
// ===== library: MasterCopy "DCS3" =====

VAR_GLOBAL   // PLC tag table "Default tag table"
   "Tag_1" AT %IW64 : Word;
   "Tag_2" AT %IW0 : Word;
   "Tag_3" AT %QW0 : Word;
   "TP_start" AT %I7.3 : Bool;
   "TP_stop" AT %I7.4 : Bool;
   "Fire" AT %I7.5 : Bool;
   "To_open_valve" AT %I7.6 : Bool;
   "Spark_on" AT %I7.7 : Bool;
   "Spark_on_1" AT %I8.0 : Bool;
   "Spark_on_2" AT %I8.1 : Bool;
   "Spark_on_3" AT %I8.2 : Bool;
   "Fire_1" AT %I8.3 : Bool;
   "Fire_2" AT %I8.4 : Bool;
   "Fire_3" AT %I8.5 : Bool;
   "Reserv_word" AT %IW68 : Word;
   "MB_Start" AT %I8.6 : Bool;   // false
   "MB_Stop" AT %I9.1 : Bool;
   "Sim_man" AT %I9.2 : Bool;
   "Sim_P_gaz_low" AT %I9.3 : Bool;
   "Sim_ACP_in" AT %IW70 : Word;
   "test" AT %I9.4 : Bool;
   "P_gaz_low" AT %I9.5 : Bool;
   "test_p_low" AT %I9.6 : Bool;
   "Tag_4" AT %IW96 : Word;
   "Tag_5" AT %IW98 : Word;
   "Clock_Byte" AT %MB0 : Byte;
   "Clock_10Hz" AT %M0.0 : Bool;
   "Clock_5Hz" AT %M0.1 : Bool;
   "Clock_2.5Hz" AT %M0.2 : Bool;
   "Clock_2Hz" AT %M0.3 : Bool;
   "Clock_1.25Hz" AT %M0.4 : Bool;
   "Clock_1Hz" AT %M0.5 : Bool;
   "Clock_0.625Hz" AT %M0.6 : Bool;
   "Clock_0.5Hz" AT %M0.7 : Bool;
   "System_Byte" AT %MB1 : Byte;
   "FirstScan" AT %M1.0 : Bool;
   "DiagStatusUpdate" AT %M1.1 : Bool;
   "AlwaysTRUE" AT %M1.2 : Bool;
   "AlwaysFALSE" AT %M1.3 : Bool;
END_VAR

TYPE "dt_AI"
   STRUCT
      Acp : DInt;   // Actual ADC code
      State : Word;
      Value : Real;   // Actual value (eng.units)
      Value_LastScan : Real;   // Last scan value
      K_filtr : Real := 0.0;   // Filter quoficient ( enable if K_filtr>0 )
      Circuit : Real;   // Actual current(mA)
      Voltage : Real;   // Actual vlotage (V)
      Resistance : Real;   // Input resistance (for voltage inputs)
      Scal_Max_Eu : Real := 100.0;   // Max scale value (eng.units)
      Scal_Min_Eu : Real := 0.0;   // Min scale value (eng.units)
      HH_Lim : Real := 100.0;   // HiHi alarm SP (eng.units)
      H_Lim : Real := 95.0;   // Hi warning SP (eng.units)
      L_Lim : Real := 5.0;   // Low warning SP (eng.units)
      LL_Lim : Real := 0.0;   // LowLow alarm SP (eng.units)
      HH_DeadBand : Real;   // HiHi alarm deadband
      H_DeadBand : Real;   // Hi warning deadband
      L_DeadBand : Real;   // Low warning deadband
      LL_DeadBand : Real;   // LowLow alarm deadband
      HH_Delay : Time;   // HiHi alarm SP delay
      H_Delay : Time;   // Hi warning SP delay
      L_Delay : Time;   // Low warning SP delay
      LL_Delay : Time;   // LowLow alarm SP delay
      Sim_Value : Real;   // Simulate value (eng.units)
      Sim_En : Bool := FALSE;   // Enable simulate mode
      Scal_Max_Upper : Bool;   // Flag Hi scale overflow
      Scal_Min_Under : Bool;   // Flag Low scale underflow
      Scale_0_20mA : Bool := FALSE;   // True - 0-20 mA, False - 4-20 mA
      Input_4mA_on_0_20mA : Bool := TRUE;   // True - 4-20mA sensor on 0-20mA current input
      VoltageInputType : Bool := FALSE;   // True -- voltage inpit, False - circuit input
      HH_Alarm : Bool;   // HiHi alarm flag
      H_Alarm : Bool;   // Hi warning flag
      L_Alarm : Bool;   // Low warning flag
      LL_Alarm : Bool;   // LowLow alarm flag
      HH_Alarm_En : Bool := TRUE;   // Enable HiHi alarm
      H_Alarm_En : Bool := FALSE;   // Enable Hi warning
      L_Alarm_En : Bool := FALSE;   // Enable Low warning
      LL_Alarm_En : Bool := TRUE;   // Enable LowLow alarm
      Short_Circuit : Bool;   // Shortcut flag
      Break : Bool;   // Breakoff flag
      Chan_Fail : Bool;   // Channel fault flag
      HH_Alarm_Logic : Bool;   // HiHi alarm for logic
      H_Alarm_Logic : Bool;   // Hi warning for logic
      L_Alarm_Logic : Bool;   // Low warning for logic
      LL_Alarm_Logic : Bool;   // LowLow alarm for logic
      Chan_Fail_Logic : Bool;   // Channel fault for logic
      Mask_mode : Bool;
      Test_mode : Bool;
      Ack_HH : Bool;
      Ack_H : Bool;
      Ack_L : Bool;
      Ack_LL : Bool;
      State_color : Byte;   // for HMI
      Ack_Alarm : Byte;   // for HMI
      Ack_Warning : Byte;   // for HMI
   END_STRUCT;
END_TYPE

TYPE "dt_DI"
   STRUCT
      Input_En : Word;
      Filter_En : Word;
      Invert_En : Word;
      Sim_En : Word;
      Sim_Value : Word;
      Input : Word;
      Value : Word;
      Value_Last_Scan : Word;
      Pins : Array[0..15] of Bool;
   END_STRUCT;
END_TYPE

TYPE "dt_DO"
   STRUCT
      Data_to_out : Byte;
      Pins : Array[0..7] of Bool;
      UsePinsAsInput : Bool;
      Invert_En : Byte;
      Output_En : Byte;
      Sim_En : Byte;
      Sim_Value : Byte;
      Value : Byte;
   END_STRUCT;
END_TYPE

DATA_BLOCK "Temp_gorelka"   // DB1
{ S7_Optimized_Access := 'FALSE' }
NAME : Scan_AI
VERSION : 1.2
// stored: InstanceOfName Scan_AI
"Scan_AI"
BEGIN
END_DATA_BLOCK

DATA_BLOCK "DI16"   // DB2
{ S7_Optimized_Access := 'FALSE' }
NAME : ScanDI16
VERSION : 1.2
// stored: InstanceOfName Scan_DI16
"Scan_DI16"
BEGIN
END_DATA_BLOCK

DATA_BLOCK "DO16"   // DB3
{ S7_Optimized_Access := 'TRUE' }
NAME : PutDO16
VERSION : 1.0
// stored: InstanceOfName Put_DO16
"Put_DO16"
BEGIN
END_DATA_BLOCK

DATA_BLOCK "Torche_DB"   // DB4
{ S7_Optimized_Access := 'FALSE' }
NAME : Torche
VERSION : 0.2
// stored: InstanceOfName Torche
"Torche"
BEGIN
END_DATA_BLOCK

DATA_BLOCK "Converse_time"   // DB6
{ S7_Optimized_Access := 'TRUE' }
VERSION : 0.1
   VAR
      Time_1 : Time;
      Time_2 : Time;
   END_VAR
BEGIN
END_DATA_BLOCK

DATA_BLOCK "temp_gorelka_2"   // DB8
{ S7_Optimized_Access := 'FALSE' }
NAME : Scan_AI
VERSION : 1.2
// stored: InstanceOfName Scan_AI
"Scan_AI"
BEGIN
END_DATA_BLOCK

DATA_BLOCK "PN_XCHANGE_DB"   // DB25
{ S7_Optimized_Access := 'FALSE' }
VERSION : 0.1
   VAR
      AI1_Ch1 : "dt_AI";   // PT200
      AI1_Ch2 : "dt_AI";   // TT200
      AI1_Ch3 : "dt_AI";   // LT200_1
      AI1_Ch4 : "dt_AI";   // LT200_2
      AI1_Ch5 : "dt_AI";   // LT201_1
      AI1_Ch6 : "dt_AI";   // LT201_2
      AI1_Ch7 : "dt_AI";   // LT202_1
      AI1_Ch8 : "dt_AI";   // LT202_2
      DI_1 : "dt_DI";   // DI CPU module
      DO_1 : "dt_DO";   // DO CPU module
   END_VAR
BEGIN
END_DATA_BLOCK

// folder: Modbus

DATA_BLOCK "Modbus_Buffer"   // DB5
{ S7_Optimized_Access := 'FALSE' }
VERSION : 0.1
   VAR
      Number_Regim : Int;   // Номер режима работы
      Alarm_number : Int;   // Номер аварии
      Time_Venting : Int;   // Время продувки факела (сек)
      Time_firing : Int;   // Время розжига факела (сек)
      Time_spark_on : Int;   // Время подачи искры во время розжига (сек)
      Time_spark_off : Int;   // Время неподачи искры (сек)
      Time_stabil : Int;   // Время стабилизации пламени (сек)
      Time_after_alarm : Int;   // Время после аварии в течении которого не учитывается наличие пламени (сек)
      Time_after_stop : Int;   // Время аварийного останова (сек)
      Time_rezerv : Int;
      Valve_to_open_lamp_on : Bool;   // Команда клапан открыт (он же состояние)
      Lamp_P_Zapal_low : Bool;   // Низкое давление газа в запальной линии
      Spark_1_to_on : Bool;   // Подача искры на свечу
      Lamp_1_on_door : Bool;   // Факел горит
      Start : Bool;   // Запустить факел (в режиме автомат)
      Stop : Bool;   // Остановить факел (в режиме автомат)
      DO_Alarm : Bool;   // Обобщенный флаг аварии
      Man_on : Bool;   // Режим факела: ручной (True - ручной, False - автомат)
      Accept_write : Bool;   // Команда на подтверждение записи
      Temp_curr_voltage : Bool;   // True -- voltage inpit, False - circuit input
      rezerv_4 : Bool;
      rezerv_5 : Bool;
      rezerv_6 : Bool;
      rezerv_7 : Bool;
      rezerv_8 : Bool;
      rezerv_9 : Bool;
      Int_rezerv : Int;
      Temp_Fire : Real;   // Температура индикации горения факела
      Temp_Fire_2 : Real;   // Температура индикации горения факела
      Scal_min : Real;   // Макс. значение инж. шкалы температуры
      Scal_min_2 : Real;   // Макс. значение инж. шкалы температуры
      Scal_max : Real;   // Мин. значение инж. шкалы температуры
      Scal_max_2 : Real;   // Мин. значение инж. шкалы температуры
      Temp_ACP : DInt;   // Значение ACP кода на датчике температуры
      Temp_ACP_2 : DInt;   // Значение ACP кода на датчике температуры
   END_VAR
BEGIN
END_DATA_BLOCK

DATA_BLOCK "MB_Parameters"   // DB11
{ S7_Optimized_Access := 'TRUE' }
VERSION : 0.1
   VAR
      MB_Load_req : Bool;
      MP_Load_Port : Port;
      MB_Load_Baud : UDInt;
      MB_Load_Parity : UInt;
      MB_Load_Done : Bool;
      MB_Load_Error : Bool;
      MB_Load_Status : Word;
      MB_Addr : UInt;
      MB_NDR : Bool;
      MB_DR : Bool;
      MB_Error : Bool;
      MB_Status : Word;
      MB_Master_req : Bool;
      MB_Master_addr : UInt;
      MB_Master_Mode : USInt;
      MB_Master_Data_addr : UDInt;
      MB_Master_Data_len : UInt;
      MB_Master_Done : Bool;
      MB_Master_Busy : Bool;
      MB_Master_Error : Bool;
      MB_Master_Status : Word;
   END_VAR
BEGIN
END_DATA_BLOCK

// folder: PROFINET

DATA_BLOCK "GeneralData"   // DB24
{ S7_Optimized_Access := 'TRUE' }
VERSION : 0.1
   VAR
      sendReq : Bool;
      contSend : Bool;
      connectSend : TCON_IP_RFC;
      doneSend : Bool;
      busySend : Bool;
      errorSend : Bool;
      statusSend : Word;
      statusSendSave : Word;
      enable : Bool;
      contRcv : Bool;
      connectRcv : TCON_IP_RFC;
      doneRcv : Bool;
      errorRcv : Bool;
      busyRcv : Bool;
      statusRcv : Word;
      statusRcvSave : Word;
      rcvdLen : UDInt;
      rcvdLenSave : UDInt;
   END_VAR
BEGIN
   connectSend.InterfaceId := 64;
   connectSend.ID := 16#9;
   connectSend.RemoteAddress.ADDR[1] := 192;
   connectSend.RemoteAddress.ADDR[2] := 168;
   connectSend.RemoteAddress.ADDR[3] := 0;
   connectSend.RemoteAddress.ADDR[4] := 8;
   connectSend.RemoteTSelector.TSelLength := 3;
   connectSend.RemoteTSelector.TSel[1] := 16#1;
   connectSend.RemoteTSelector.TSel[2] := 16#2;
   connectSend.RemoteTSelector.TSel[3] := 16#3;
   connectSend.LocalTSelector.TSelLength := 3;
   connectSend.LocalTSelector.TSel[1] := 16#1;
   connectSend.LocalTSelector.TSel[2] := 16#2;
   connectSend.LocalTSelector.TSel[3] := 16#3;
   connectRcv.InterfaceId := 64;
   connectRcv.ID := 16#10;
   connectRcv.RemoteAddress.ADDR[1] := 192;
   connectRcv.RemoteAddress.ADDR[2] := 168;
   connectRcv.RemoteAddress.ADDR[3] := 0;
   connectRcv.RemoteAddress.ADDR[4] := 8;
   connectRcv.RemoteTSelector.TSelLength := 4;
   connectRcv.RemoteTSelector.TSel[1] := 16#1;
   connectRcv.RemoteTSelector.TSel[2] := 16#2;
   connectRcv.RemoteTSelector.TSel[3] := 16#3;
   connectRcv.LocalTSelector.TSelLength := 4;
   connectRcv.LocalTSelector.TSel[1] := 16#1;
   connectRcv.LocalTSelector.TSel[2] := 16#2;
   connectRcv.LocalTSelector.TSel[3] := 16#3;
   connectRcv.RemoteTSelector.TSel[4] := 16#4;
   connectRcv.LocalTSelector.TSel[4] := 16#4;
END_DATA_BLOCK

// folder: (top level)

FUNCTION_BLOCK "Torche"   // FB8, SCL
TITLE = Torche (current control)
{ S7_Optimized_Access := 'FALSE' }
NAME : Torche
VERSION : 0.2
   VAR_INPUT
      Man_fakel : Bool;
      Fakel_fire_is_on : Bool;
      Temp_rozgik_FND_1 : Bool;
      Temp_rozgik_FND_2 : Bool;
      Temp_rozgik_FVD_1 : Bool;
      Temp_rozgik_FVD_2 : Bool;
      P_gaz_low : Bool;
      Frequency_1_in_mode : Bool := 0;
      Frequency_2_in_mode : Bool := 0;
      Frequency_1_Fail : Word := 0;
      Frequency_2_Fail : Word := 0;
      Frequency_1_State : Word := 0;
      Frequency_2_State : Word := 0;
      Flow_Low : Bool;
      Flow_Lo_FND : Bool;
      Flow_Lo_FVD : Bool;
      Panel_vent_1_off : Bool;
      Panel_vent_1_on : Bool;
      Panel_vent_2_off : Bool;
      Panel_vent_2_on : Bool;
      Stop : Bool;
      Start : Bool;
      Valve_to_open_man : Bool;
      Timer_start_FND : Bool;
      Timer_start_FVD : Bool;
   END_VAR
   VAR_OUTPUT
      Number_regim : Int;
      DO_Alarm : Bool;
      Alarm_number : Int;
      Frequency_1_Cmd_on : Word;
      Frequency_2_Cmd_on : Word;
      Valve_to_open : Bool;
      Lamp_on_valve_open : Bool;
      Lamp_P_zapal_low : Bool;
      Spark_1_to_on : Bool;
      Spark_2_to_on : Bool;
      Spark_3_to_on : Bool;
      Spark_4_to_on : Bool;
      Start_algoritm_gaz_vozduh_1 : Bool;
      Start_algoritm_gaz_vozduh_2 : Bool;
      Frequency_1_Cmd_off : Word;
      Frequency_2_Cmd_off : Word;
      Frequency_1_Cmd_Reset_Error : Word;
      Frequency_2_Cmd_Reset_Error : Word;
      Lamp_1_on_door : Bool;
      Fire_is_off_1 : Bool;
      Lamp_2_on_door : Bool;
      Fire_is_off_2 : Bool;
   END_VAR
   VAR
      Signal_Torche : Struct
         Vers_number : Int;
         Frequency_1_Mode : Word;
         Frequency_2_Mode : Word;
         Man_auto : Bool;
         ANY_Stop_fakel : Bool;
         Warning_bool_1 : Bool;
         Warning_bool_2 : Bool;
         Warning_bool_3 : Bool;
         Warning_bool_4 : Bool;
         Warning_bool_5 : Bool;
         Warning_bool_6 : Bool;
         Warning_bool_7 : Bool;
         Warning_bool_8 : Bool;
         Warning : Bool;
         Alarm_bool_1 : Bool;
         Alarm_bool_2 : Bool;
         Alarm_bool_3 : Bool;
         Alarm_bool_4 : Bool;
         Alarm_bool_5 : Bool;
         Alarm_state : Bool;
         Stop_vent_1 : Bool;
         Stop_vent_2 : Bool;
         Start_vent_1 : Bool;
         Start_vent_2 : Bool;
         ANY_Klapan_time : Bool;
         Privod_not_load : Bool;
         ANY_Start_timer : Bool;
         ANY_Start_rozgik : Bool;
         ANY_bool_1 : Bool;
         ANY_bool_2 : Bool;
         pererozgig : Bool;
         ANY_Time_stabil : Bool;
         Rezerv_Alarmstop_on : Bool;
         ANY_Time_after_alarms : Bool;
         Time_after_alm_g : Int;
         Time_stabiliz_g : Int;
         Time_firing_g : Int;
         Time_vent_g : Int;
         Time_stop_fire_g : Int;
         Time_start_g : Int;
         Time_klapan : Int;
         Time_fire_off_g : Int;
         Time_spark_off_g : Int;
         Time_spark_on_g : Int;
         Time_after_alm_t : Time;
         Time_stabiliz_t : Time;
         Time_firing_t : Time;
         Time_vent_t : Time;
         Time_stop_fire_t : Time;
         Time_start_t : Time;
         Time_fire_off_t : Time;
         Time_spark_off_t : Time;
         Time_spark_on_t : Time;
         Venting_start : Bool;
         Valve_opening_start : Bool;
         Sparking_start : Bool;
         Stabilization_start : Bool;
         After_alarm_start : Bool;
         After_stop_start : Bool;
         Spark_off_start : Bool;
         Spark_on_start : Bool;
         Fire_time_1 : Bool;
      END_STRUCT;
      Venting : TON_TIME;
      Valve_opening : TON_TIME;
      Sparking : TON_TIME;
      Stabilization : TON_TIME;
      After_alarm : TON_TIME;
      After_stop : TON_TIME;
      Spark_off : TON_TIME;
      Spark_on : TOF_TIME;
   END_VAR
BEGIN

   (*
   Блок предназначен для управления двумя версиями факела (#Signal_Torche.Vers_number - номера версии прошивки факелов). В данном варианте у нас 1-я версия факела, простая версия.

   Факела запускается только в режиме автомат (#Man_fakel = false) при нажатии #Start. При нажатии #Stop факел выходит в 0-ой режим из любого состояния.

   У факела существует 7 режимов (#Number_regim) Готовность, запуск частотных приводов (во 2-ой версии прошивки факела) продувка, розжиг, 
   стабилизация, автоматический режим (нормальный режим работы факела в автомате), аварийный стоп.
   *)


   //***********************************************************Таймера***********************
   //***********Таймер  отсутствия обработки аварии после останова факела**************
   #After_stop(IN := #Signal_Torche.After_stop_start // IN: BOOL
               ,
               PT := #Signal_Torche.Time_stop_fire_t// IN: TIME
   );
   //***********Таймер розжига факела**************
   #Sparking(IN := #Signal_Torche.Sparking_start // IN: BOOL
             ,
             PT := #Signal_Torche.Time_firing_t// IN: TIME
   );
   //***********Таймер отсутствия искры при розжиге**************
   #Spark_off(IN := #Signal_Torche.Spark_off_start // IN: BOOL
              ,
              PT := #Signal_Torche.Time_spark_off_t// IN: TIME
   );

   //***********Таймер наличия искры при розжиге**************
   #Spark_on(IN := #Signal_Torche.Spark_on_start // IN: BOOL
             ,
             PT := #Signal_Torche.Time_spark_on_t// IN: TIME
   );

   //***********Таймер нахождения в аварийном состоянии**************
   #After_alarm(IN := #Signal_Torche.After_alarm_start // IN: BOOL
                ,
                PT := #Signal_Torche.Time_after_alm_t// IN: TIME
   );

   //***********Таймер стабилизации пламени**************
   #Stabilization(IN := #Signal_Torche.Stabilization_start // IN: BOOL
                  ,
                  PT := #Signal_Torche.Time_stabiliz_t// IN: TIME
   );

   //***********Таймер продувки факела**************
   #Venting(IN := #Signal_Torche.Venting_start // IN: BOOL
            ,
            PT := #Signal_Torche.Time_vent_t // IN: TIME
   );

   #Signal_Torche.Time_vent_t := T_CONV(#Signal_Torche.Time_vent_g)*1000;
   #Signal_Torche.Time_stop_fire_t := T_CONV(#Signal_Torche.Time_stop_fire_g)*1000;
   #Signal_Torche.Time_firing_t := T_CONV(#Signal_Torche.Time_firing_g)*1000;
   #Signal_Torche.Time_stabiliz_t := T_CONV(#Signal_Torche.Time_stabiliz_g)*1000;
   #Signal_Torche.Time_spark_off_t := T_CONV(#Signal_Torche.Time_spark_off_g)*1000;
   #Signal_Torche.Time_spark_on_t := T_CONV(#Signal_Torche.Time_spark_on_g)*1000;
   #Signal_Torche.Time_after_alm_t :=T_CONV(#Signal_Torche.Time_after_alm_g)*1000;

   //если факел не в режиме ручной
   IF NOT #Man_fakel THEN 

       IF #Signal_Torche.Vers_number = 2 THEN
           #Signal_Torche.Frequency_1_Mode := 8;
           #Signal_Torche.Frequency_2_Mode := 8;
       END_IF;

     #Signal_Torche.Man_auto := false;
     CASE #Number_regim OF
       0:

         (*IF  Temp_TON_2_ET = T#0s   THEN
              IF Valve_Open = true THEN   
                  Lamp_on_valve_open := true;
                  Warning_bool_1 := true;
              ELSE
                  Lamp_on_valve_open := false;
                  Warning_bool_1 := false;
              END_IF;

          ELSIF Temp_TON_2_ET > T#0s and Temp_TON_2_ET < Timer_2  THEN
              Warning_bool_1 := false;            
          ELSIF TEMP_TON_2_Q THEN 
              ANY_Klapan_time := false;

          END_IF;*)




           //Таймер после останова факела, для времени остывания факела и невыдачи в это время Warning
           IF #After_stop.ET = T#0s THEN //если таймер не вкл

                IF ((#Signal_Torche.Vers_number = 1) AND (#Fakel_fire_is_on = true)) OR ((#Signal_Torche.Vers_number = 2) AND ((#Temp_rozgik_FND_1 = true) OR (#Temp_rozgik_FND_2 = true) OR (#Temp_rozgik_FVD_1 = true) OR (#Temp_rozgik_FVD_2 = true))) THEN

                   #Signal_Torche.Warning_bool_2 := true;
             (*IF   Vers_number = 2 and not (Flow_Lo_FND or Flow_Lo_FVD) THEN 
                    Warning_bool_5 := true;
                ELSE
                    Warning_bool_5 := FALSE;
                END_IF;*)

                ELSE

               #Signal_Torche.Warning_bool_2 := false;
             (*IF    Vers_number = 2 and not (Flow_Lo_FND or Flow_Lo_FVD) THEN 
                 Warning_bool_6 := true;
             ELSE
                 Warning_bool_6 := FALSE;
             END_IF;*)
                END_IF;

           ELSIF #After_stop.ET > T#0s AND #After_stop.ET < T#600s THEN //если таймер запущен
             #Signal_Torche.Warning_bool_2 := false;
             #Signal_Torche.Warning_bool_6 := false;
         END_IF;
         IF #After_stop.Q THEN  //если таймер прошел заданное время - сбрасываем его
             #Signal_Torche.Warning_bool_8 := false;
             #Signal_Torche.After_stop_start := false;
         END_IF;



         IF #P_gaz_low THEN //если низкое давление газа
             #Signal_Torche.ANY_Stop_fakel := true;
         ELSE
             #Signal_Torche.ANY_Stop_fakel := false;
         END_IF;

         IF #Signal_Torche.Vers_number = 2 THEN//Версия прошивки №2


           IF #Frequency_1_in_mode OR #Frequency_2_in_mode THEN// если режим частотного привода ручной
               #Signal_Torche.Warning_bool_3 := true;//поджигаем аварию
           ELSE
               #Signal_Torche.Warning_bool_3 := false;
           END_IF;



           (*IF (Frequency_1_Fail <> 0) or (Frequency_2_Fail <> 0) THEN
               Warning_bool_4 := true;
           ELSE
               Warning_bool_4 := false;
           END_IF;*)
         END_IF;


        //**формирование единого флага "Предупреждение"
         IF #Signal_Torche.Warning_bool_1 OR #Signal_Torche.Warning_bool_2 OR #Signal_Torche.Warning_bool_3 OR #Signal_Torche.Warning_bool_4 OR #Signal_Torche.Warning_bool_5 OR #Signal_Torche.Warning_bool_6 OR #Signal_Torche.Warning_bool_7 OR #Signal_Torche.ANY_Stop_fakel THEN
             #Signal_Torche.Warning := true;
         ELSE
             #Signal_Torche.Warning := false;
         END_IF;



         IF #Signal_Torche.Vers_number = 2 THEN

           (*IF  Press_razryagenie_FND or Press_razryagenie_FVD  THEN
               Alarm_bool_1 := true;
           ELSE
               Alarm_bool_1 := false;
           END_IF;*)


           IF #Frequency_1_Fail <> 0 OR #Frequency_2_Fail <> 0 THEN
               #Signal_Torche.Alarm_bool_2 := true;
           ELSE
               #Signal_Torche.Alarm_bool_2 := false;

           END_IF;
           //**формирование единого флага "Авария"
           IF #Signal_Torche.Alarm_bool_1 OR #Signal_Torche.Alarm_bool_2 OR #Signal_Torche.Alarm_bool_3 OR #Signal_Torche.Alarm_bool_4 OR #Signal_Torche.Alarm_bool_5 THEN
               #Signal_Torche.Alarm_state := true;
             #DO_Alarm := true;
           ELSE
               #Signal_Torche.Alarm_state := false;
             #DO_Alarm := false;
           END_IF;


         END_IF;


         #Signal_Torche.Stop_vent_1 := false;

         #Signal_Torche.Stop_vent_2 := false;

         #Signal_Torche.Start_vent_1 := false;

         #Signal_Torche.Start_vent_2 := false;


         IF #Start AND NOT #P_gaz_low THEN

           //Обработка запуска при версии прошивки 2
             IF #Signal_Torche.Vers_number = 2 THEN
                 IF NOT #Signal_Torche.Alarm_state = true THEN
               #Alarm_number := 0;
               #Number_regim := 11;
               #Signal_Torche.Stop_vent_1 := true;
               #Signal_Torche.Stop_vent_2 := true;
           END_IF;
           //Обработка запуска при версии прошивки 1
         ELSIF #Signal_Torche.Vers_number = 1 THEN
             #Alarm_number := 0;
             #Number_regim := 1;
           END_IF;
           #Signal_Torche.Warning := false;
           #Signal_Torche.ANY_Klapan_time := false;
           #Signal_Torche.Warning_bool_8 := false;
           #Signal_Torche.After_stop_start := false;

         END_IF;





     11: // *****************************Режим включения приводов*********************

         IF #Frequency_1_Fail = 0 AND #Frequency_2_Fail = 0 THEN // нет ошибок приводов
           IF NOT (#Timer_start_FND) AND #Frequency_1_State = 0 THEN // Привод на Факел низкого давления выключен и не запускается
             #Frequency_1_Cmd_on := 8; // Запускаем его
           END_IF;
           IF NOT (#Timer_start_FVD) AND #Frequency_2_State = 0 THEN// Привод на Факел высокого давления выключен и не запускается
               #Frequency_2_Cmd_on := 8;// Запускаем его
           END_IF;
           IF #Frequency_1_State = 1 AND #Frequency_2_State = 1 THEN // ОБА Привода включены
               IF #Signal_Torche.Privod_not_load = true THEN //Мы пришли сюда из 4-го режима (автоматическая работа) по причине выключения одного из приводов
               #Number_regim := 4; // переходим в режим 4
               #Signal_Torche.Privod_not_load := false;
             ELSE
                 #Number_regim := 1;  // переходим в режим 1
               #Signal_Torche.Stop_vent_1 := false;
               #Signal_Torche.Stop_vent_2 := false;
             END_IF;
           END_IF;
         ELSIF #Frequency_1_Fail <> 0 OR #Frequency_2_Fail <> 0 THEN //Ошибка на одном из приводов
             IF #Signal_Torche.Privod_not_load = true THEN//Мы пришли сюда из 4-го режима (автоматическая работа) по причине выключения одного из приводов
                 #Number_regim := 4; // переходим в режим 4 с предупреждением
             #Signal_Torche.Warning := true;
             #Frequency_1_Cmd_on := 0;
             #Frequency_2_Cmd_on := 0;
         ELSE // Уходим в режим готовность с необходимой аварией
             #Valve_to_open := false;
             #Lamp_on_valve_open := false;
               #Signal_Torche.Alarm_state := true;
             #DO_Alarm := true;
             #Number_regim := 0;
             #Signal_Torche.Stop_vent_1 := false;
             #Signal_Torche.Stop_vent_2 := false;
             #Alarm_number := 111;(*------------------------------------------------------------------------------------*)
             #Frequency_1_Cmd_on := 0;
             #Frequency_2_Cmd_on := 0;
           END_IF;
         END_IF;


     1: // *****************************Режим продувки*********************
         IF NOT #P_gaz_low THEN // нет низкого давления газа в запальной линии
   //***********************************************// если версия прошивки 2 *******************************************************************************************************

             IF #Signal_Torche.Vers_number = 2 THEN
           (*IF (Razryag_line_1 or Razryag_line_2) THEN
               Alarm_number :=  12; 
               Number_regim := 5;
               ANY_Klapan_time := false;
               ANY_Start_timer := false;
           END_IF;*)

            IF (#Signal_Torche.Vers_number = 2) AND (#Frequency_1_Fail <> 0 OR #Frequency_2_Fail <> 0) THEN
               #Alarm_number := 13; (*--------------------------------------ошибка приводов----------------------------------------------*)
               #Number_regim := 5;
               #Valve_opening.IN := false;
               #Signal_Torche.Venting_start := false;
           END_IF;
             IF (#Signal_Torche.Vers_number = 2) AND (#Signal_Torche.Frequency_1_Mode <> 8 OR #Signal_Torche.Frequency_2_Mode <> 8) THEN
               #Alarm_number := 14; (*-----------------------------------Неправильный режим работы приводов-------------------------------------------------*)
               #Number_regim := 5;
               #Valve_opening.IN := false;
               #Signal_Torche.Venting_start := false;
           END_IF;
             IF (#Temp_rozgik_FND_1 OR #Temp_rozgik_FND_2 OR #Temp_rozgik_FVD_1 OR #Temp_rozgik_FVD_2) AND #Flow_Low THEN
               #Alarm_number := 15; (*----------------------------------Расход в основной линии и высокая температура на факеле--------------------------------------------------*)
               #Number_regim := 5;
               #Valve_opening.IN := false;
               #Signal_Torche.Venting_start := false;
           END_IF;
             IF NOT (#Flow_Low) THEN
                 #Alarm_number := 16; (*----------------------------------- Расход в основной линии -------------------------------------------------*)
               #Number_regim := 5;
               #Valve_opening.IN := false;
               #Signal_Torche.Venting_start := false;
             END_IF;
             IF (#Frequency_1_State <> 1) OR (#Frequency_2_State <> 1) THEN
                 #Alarm_number := 18; (*--------------------------------------один из  приводов выключен----------------------------------------------*)
               #Number_regim := 5;
               #Valve_opening.IN := false;
               #Signal_Torche.Venting_start := false;
             END_IF;
           END_IF;
   //*****************************************************************************************************************************************************************************




           #Valve_to_open := TRUE; // открываем клапан

           (* #Valve_opening.IN := true*)

           (*IF #Valve_opening.Q THEN *)
           #Lamp_on_valve_open := true; 
           (*  #Valve_opening.IN := false;*)
           #Signal_Torche.Venting_start := true; // включаем таймер на продувку
           (*#Venting(IN := #Signal_Torche.Venting_start // IN: BOOL
                    ,
                    PT := #Signal_Torche.Time_vent_t // IN: TIME
           );*)
           IF (#Venting.Q) THEN (*(TEMP_TON_1_Q and (NOT TEMP_TON_2_Q))*) // если таймер прошел - переходим в режим 2
             #Number_regim := 2;
             #Signal_Torche.Venting_start := false;
           END_IF;
           (*ELSIF (NOT Valve_Open and (#Valve_opening.Q ))  THEN                       
                     Alarm_number :=  11;
                     Number_regim := 0;
                     ANY_Klapan_time := false;
                     ANY_Start_timer := false;
           END_IF;     *)
          ELSE
             IF #P_gaz_low THEN // низкое давления газа в запальной линии
             #Lamp_P_zapal_low := true;
           END_IF;


           #Alarm_number := 10;(*-----------------------------------Отключаем все таймеры, ставим нужный аларм-------------------------------------------------*)
           #Valve_opening.IN  := false;
           #Signal_Torche.Venting_start := false;
           #Valve_to_open := false;
           #Lamp_on_valve_open := false;
           IF #Signal_Torche.Vers_number = 2 THEN
             #Number_regim := 5;
             ELSIF #Signal_Torche.Vers_number = 1 THEN
             #Number_regim := 0;
           END_IF;
         END_IF;
     2: // *****************************Режим розжига*********************
         IF NOT #P_gaz_low THEN
         (*IF not Valve_Open THEN
             Alarm_number := 27;
             Lamp_on_valve_open := false;            
             Number_regim := 5;
             ANY_Start_rozgik := false;
             ANY_bool_1 := false;
             ANY_bool_2 := false;
             Spark_1_to_on := false;
             pererozgig := FALSE;
             Warning := FALSE;               
         END_IF;*)
    //***********************************************// если версия прошивки 2 *******************************************************************************************************

             IF #Signal_Torche.Vers_number = 2 THEN
                 IF (#Signal_Torche.Vers_number = 2) AND (#Frequency_1_Fail <> 0 OR #Frequency_2_Fail <> 0) THEN
               #Alarm_number := 23; (*------------------------------------------------------------------------------------*)
               #Number_regim := 5;
               #Signal_Torche.Sparking_start := false;
               #Signal_Torche.Spark_on_start := false;
               #Signal_Torche.Spark_off_start := false;
               #Spark_1_to_on := false;
               #Spark_2_to_on := false;
               #Spark_3_to_on := false;
               #Spark_4_to_on := false;
               #Signal_Torche.pererozgig := FALSE;
               #Signal_Torche.Warning := FALSE;
             END_IF;
             IF (#Signal_Torche.Vers_number = 2) AND (#Signal_Torche.Frequency_1_Mode <> 8 OR #Signal_Torche.Frequency_2_Mode <> 8) THEN
               #Alarm_number := 24; (*------------------------------------------------------------------------------------*)
               #Number_regim := 5;
               #Signal_Torche.Sparking_start := false;
               #Signal_Torche.Spark_on_start := false;
               #Signal_Torche.Spark_off_start := false;
               #Spark_1_to_on := false;
               #Spark_2_to_on := false;
               #Spark_3_to_on := false;
               #Spark_4_to_on := false;
               #Signal_Torche.pererozgig := FALSE;
               #Signal_Torche.Warning := FALSE;
             END_IF;
             IF NOT (#Flow_Low) THEN
               #Alarm_number := 26;    (*------------------------------------------------------------------------------------*)
               #Number_regim := 5;
               #Signal_Torche.Sparking_start := false;
               #Signal_Torche.Spark_on_start := false;
               #Signal_Torche.Spark_off_start := false;
               #Spark_1_to_on := false;
               #Spark_2_to_on := false;
               #Spark_3_to_on := false;
               #Spark_4_to_on := false;
               #Signal_Torche.pererozgig := FALSE;
               #Signal_Torche.Warning := FALSE;
             END_IF;
             IF (#Frequency_1_State <> 1) OR (#Frequency_2_State <> 1) THEN
               #Alarm_number := 28; (*------------------------------------------------------------------------------------*)
               #Number_regim := 5;
               #Signal_Torche.Sparking_start := false;
               #Signal_Torche.Spark_on_start := false;
               #Signal_Torche.Spark_off_start := false;
               #Spark_1_to_on := false;
               #Spark_2_to_on := false;
               #Spark_3_to_on := false;
               #Spark_4_to_on := false;
               #Signal_Torche.pererozgig := FALSE;
               #Signal_Torche.Warning := FALSE;
             END_IF;
         END_IF;
   //******************************************************************************************************************************************** ************************************* 

         #Signal_Torche.Sparking_start := true; //запускаем таймер на розжиг
         (*#Sparking(IN := #Signal_Torche.Sparking_start // IN: BOOL
                  ,
                  PT := #Signal_Torche.Time_firing_t // IN: TIME
         );
         *)

         IF NOT #Sparking.Q THEN // если таймер на розжиг не прошел то включаем/выключаем искру периодически
             #Signal_Torche.Spark_off_start := #Spark_on.Q;
             #Signal_Torche.Spark_on_start := NOT #Spark_off.Q;
             (*
            #Spark_off(IN := #Signal_Torche.Spark_off_start// IN: BOOL
                       ,
                       PT := #Signal_Torche.Time_spark_off_t // IN: TIME
            );

            #Spark_on(IN := #Signal_Torche.Spark_on_start // IN: BOOL
                       ,
                       PT := #Signal_Torche.Time_spark_on_t // IN: TIME
            );
            *)
           (*ANY_bool_1 := TEMP_TOF_1_Q;
           ANY_bool_2 := NOT TEMP_TON_4_Q;*)
               IF #Spark_off.Q THEN // таймер на выключение искры
                   IF #Signal_Torche.Vers_number = 2 THEN
                 #Spark_1_to_on := true;
                 #Spark_2_to_on := true;
                 #Spark_3_to_on := true;
                 #Spark_4_to_on := true;
                   ELSIF #Signal_Torche.Vers_number = 1 THEN
                 #Spark_1_to_on := true;
               END_IF;
             END_IF;
             IF NOT #Spark_off.Q THEN // таймер на включение искры
                 IF #Signal_Torche.Vers_number = 2 THEN
                 #Spark_1_to_on := false;
                 #Spark_2_to_on := false;
                 #Spark_3_to_on := false;
                 #Spark_4_to_on := false;
                 ELSIF #Signal_Torche.Vers_number = 1 THEN
                 #Spark_1_to_on := false;
               END_IF;
             END_IF;


         ELSIF #Sparking.Q THEN // если таймер прошел - переходим в режим стабилизации (ожидания появления пламени)

             #Number_regim := 3; // идем в режим стабилизации предварительно отключив все таймеры и сбросив сигнал на подачу искры

             #Signal_Torche.Sparking_start := false;
             #Signal_Torche.Spark_on_start := false;
             #Signal_Torche.Spark_off_start := false;
             IF #Signal_Torche.Vers_number = 2 THEN
               #Spark_1_to_on := false;
               #Spark_2_to_on := false;
               #Spark_3_to_on := false;
               #Spark_4_to_on := false;
           ELSIF #Signal_Torche.Vers_number = 1 THEN
               #Spark_1_to_on := false;
             END_IF;

           END_IF;

           IF #Sparking.ET > T#5s AND #Fakel_fire_is_on THEN // если прошло более 5 сек розжига и появилось пламя - идем в режим 4 предварительно отключив все таймеры и сбросив сигнал на подачу искры
               #Signal_Torche.Sparking_start := false;
               #Signal_Torche.Spark_on_start := false;
               #Signal_Torche.Spark_off_start := false;

             #Spark_1_to_on := false;
             #Spark_2_to_on := false;
             #Spark_3_to_on := false;
             #Spark_4_to_on := false;
             #Signal_Torche.pererozgig := FALSE;
             #Signal_Torche.Warning := FALSE;
             #Alarm_number := 0;
             #Number_regim := 4;

           END_IF;

         ELSE
           IF #P_gaz_low THEN
             #Lamp_P_zapal_low := true;
           END_IF;

           #Alarm_number := 20;    (*------------------------------------------------------------------------------------*)
           #Signal_Torche.Sparking_start := false;
           #Signal_Torche.Spark_on_start := false;
           #Signal_Torche.Spark_off_start := false;
           #Spark_1_to_on := false;
           #Spark_2_to_on := false;
           #Spark_3_to_on := false;
           #Spark_4_to_on := false;
           #Signal_Torche.pererozgig := FALSE;
           #Signal_Torche.Warning := FALSE;
           #Valve_to_open := false;
           #Lamp_on_valve_open := false;
           IF #Signal_Torche.Vers_number = 2 THEN
             #Number_regim := 5;
         ELSIF #Signal_Torche.Vers_number = 1 THEN
             #Number_regim := 0;
           END_IF;
         END_IF;

       3: // ****************************************режим стабилизации**********************

         IF NOT #P_gaz_low THEN
         (*IF not Valve_Open THEN
             Alarm_number := 37;
             Lamp_on_valve_open := false;            
             Number_regim := 5;
             ANY_Time_stabil := false;           
         END_IF;*)

   //***********************************************// если версия прошивки 2 *******************************************************************************************************
             IF #Signal_Torche.Vers_number = 2 THEN
                 IF (#Signal_Torche.Vers_number = 2) AND (#Frequency_1_Fail <> 0 OR #Frequency_2_Fail <> 0) THEN
               #Alarm_number := 33; (*------------------------------------------------------------------------------------*)
               #Number_regim := 5;
               #Signal_Torche.Stabilization_start := false;
             END_IF;
             IF (#Signal_Torche.Vers_number = 2) AND (#Signal_Torche.Frequency_1_Mode <> 8 OR #Signal_Torche.Frequency_2_Mode <> 8) THEN
               #Alarm_number := 34; (*------------------------------------------------------------------------------------*)
               #Number_regim := 5;
               #Signal_Torche.Stabilization_start := false;
             END_IF;

             IF NOT (#Flow_Low) THEN
               #Alarm_number := 36; (*------------------------------------------------------------------------------------*)
               #Number_regim := 5;
               #Signal_Torche.Stabilization_start := false;
               ;
             END_IF;
             IF (#Frequency_1_State <> 1) OR (#Frequency_2_State <> 1) THEN
               #Alarm_number := 38; (*------------------------------------------------------------------------------------*)
               #Number_regim := 5;
               #Signal_Torche.Stabilization_start := false;
             END_IF;
         END_IF;
   //******************************************************************************************************************************************** ************************************* 
           #Signal_Torche.Stabilization_start := true; // запускаем таймер стабилизации
           IF #Stabilization.ET > t#0s AND #Fakel_fire_is_on THEN //Если пламя во время режима стабилизации появилось - переходим в автоматический режим работы (4)
               #Signal_Torche.Stabilization_start := false;
             #Number_regim := 4;
             #Signal_Torche.pererozgig := FALSE;
             #Signal_Torche.Warning := FALSE;
             #Alarm_number := 0;(*------------------------------------------------------------------------------------*)

           ELSIF #Stabilization.Q AND NOT #Fakel_fire_is_on THEN //Если таймер прошел а пламя не появилось
             IF NOT #Signal_Torche.pererozgig THEN //если мы пришли сюда из 4-го режима (в случае потухании факела) то идем в режим 0, предварительно отключив все таймеры и выставив аларм
               #Valve_to_open := false;
               #Lamp_on_valve_open := false;
               #Signal_Torche.Stabilization_start := false;
               #Number_regim := 0;
               #Alarm_number := 31;(*------------------------------------------------------------------------------------*)
               #Signal_Torche.pererozgig := FALSE;
               #Signal_Torche.Warning := FALSE;
             ELSIF #Signal_Torche.pererozgig THEN//идем в режим 5, предварительно отключив все таймеры и выставив аларм
               #Signal_Torche.Stabilization_start := false;
               #Number_regim := 5;
               #Signal_Torche.pererozgig := FALSE;
               #Alarm_number := 41;(*------------------------------------------------------------------------------------*)
             END_IF;
           END_IF;

         ELSE
           IF #P_gaz_low THEN
             #Lamp_P_zapal_low := true;
           END_IF;
           #Alarm_number := 30;(*------------------------------------------------------------------------------------*)
           #Signal_Torche.Stabilization_start := false;
           #Valve_to_open := false;
           #Lamp_on_valve_open := false;
           IF #Signal_Torche.Vers_number = 2 THEN
             #Number_regim := 5;
           ELSIF #Signal_Torche.Vers_number = 1 THEN
             #Number_regim := 0;
           END_IF;
         END_IF;
     4: // ****************************************режим автоматической работы**********************

    //*************************************************************************// если версия прошивки 2 ****************************************************************************
           IF #Signal_Torche.Vers_number = 2 THEN 
               IF (#Signal_Torche.Frequency_1_Mode <> 8 OR #Signal_Torche.Frequency_2_Mode <> 8) THEN // режим работы приводов не авто
                   #Signal_Torche.Warning := true; // выставляем "Предупреждение"
               ELSE
                   #Signal_Torche.Warning := false;
               END_IF;

               IF (#Frequency_1_Fail <> 0 OR #Frequency_2_Fail <> 0) THEN // Появилась ошибка приводов
                   #Signal_Torche.Warning := true; // выставляем "Предупреждение"
           ELSE
               #Signal_Torche.Privod_not_load := false;
               #Signal_Torche.Warning := false;
           END_IF;
           IF (#Frequency_1_State <> 1 OR #Frequency_2_State <> 1) AND (#Signal_Torche.Privod_not_load = false) THEN  // один из приводов выключен 
               #Signal_Torche.Privod_not_load := true; // зажигаем флаг: перезапустить привода
             #Number_regim := 11; // переходим в режим : запуск приводов
             #Alarm_number := 402;(*----------------------------выставляем нужную ошибку--------------------------------------------------------*)
             #Signal_Torche.Start_vent_1 := false;
             #Signal_Torche.Start_vent_2 := false;

           END_IF;


           IF NOT #Flow_Lo_FND THEN // если в трубе на факеле  никого давления есть расход 
               #Signal_Torche.Start_vent_1 := true;  // запускаем вентиляторы для подачи воздуха
               #Start_algoritm_gaz_vozduh_1 := true; // запускаем алгоритм регулирования соотношения расхода газ/воздух
           END_IF;
           IF NOT #Flow_Lo_FVD THEN // если в трубе на факеле  высокого давления есть расход 
               #Signal_Torche.Start_vent_2 := true;
             #Start_algoritm_gaz_vozduh_2 := true;
           END_IF;

           IF #Flow_Lo_FND THEN // если в трубе на факеле  никого давления нет расход а
               #Signal_Torche.Stop_vent_1 := #Panel_vent_1_off; // возможность откл. вентилятора с БАРКП
               #Signal_Torche.Start_vent_1 := #Panel_vent_1_on; // возможность вкл. вентилятора с БАРКП
               IF #Signal_Torche.Start_vent_1 AND NOT #Signal_Torche.Stop_vent_1 THEN
               #Start_algoritm_gaz_vozduh_1 := true;
           ELSIF #Signal_Torche.Stop_vent_1 AND NOT #Signal_Torche.Start_vent_1 THEN
               #Start_algoritm_gaz_vozduh_1 := true;
             END_IF;


           END_IF;
           IF #Flow_Lo_FVD THEN // если в трубе на факеле  высокого давления нет расхода
               #Signal_Torche.Stop_vent_2 := #Panel_vent_2_off; // возможность откл. вентилятора с БАРКП
               #Signal_Torche.Start_vent_2 := #Panel_vent_2_on; // возможность вкл. вентилятора с БАРКП
               IF #Signal_Torche.Start_vent_2 AND NOT #Signal_Torche.Stop_vent_2 THEN
                   #Start_algoritm_gaz_vozduh_2 := true; // если вентилятор включен - запускаем алгоритм регулирования соотношения расхода газ/воздух
           ELSIF #Signal_Torche.Stop_vent_2 AND NOT #Signal_Torche.Start_vent_2 THEN
               #Start_algoritm_gaz_vozduh_2 := true; // если вентилятор включен - запускаем алгоритм регулирования соотношения расхода газ/воздух
             END_IF;


           END_IF;
         END_IF;

         //******************************************************************************************************************************************** ************************************* 


         IF #P_gaz_low THEN // при низком давлении газа в запальной линии - переходим в аварийное состояние
           #Alarm_number := 40;(*------------------------------------------------------------------------------------*)
           #Number_regim := 5;
           #Lamp_P_zapal_low := true;



         END_IF;





         (*IF Valve_Open = false THEN 
             Warning := true;
             Lamp_on_valve_open := false;
         else 
             Warning := false;
             Lamp_on_valve_open := true;

         END_IF;*)




         IF NOT #Fakel_fire_is_on THEN // если пропадание пламени (низкая температура у факела) - переходим в режим розжига
             #Signal_Torche.pererozgig := TRUE; // зажигаем флаг перерозжига
           #Number_regim := 2;
           #Signal_Torche.Warning := true;
           #Alarm_number := 401;(*---------------------Зажигаем аварию перерозжиг---------------------------------------------------------------*)

         END_IF;


     5:// ****************************************режим ававрийного останова**********************
         IF NOT #Signal_Torche.After_alarm_start = true THEN
             #Signal_Torche.After_alarm_start := true;// запускаем таймер аварийного останова
         END_IF;
         #Signal_Torche.Privod_not_load := false; // отключаем привода, закрываем клапан
         #Valve_to_open := false;
         #Lamp_on_valve_open := false;
         (*ANY_Klapan_time := true;*)
         #Signal_Torche.ANY_Time_after_alarms := true;
         #Signal_Torche.Alarm_state := true;
         #DO_Alarm := true;

   //***********************************************// если версия прошивки 2 *************************************      
         IF #Signal_Torche.Vers_number = 2 THEN
             #Signal_Torche.Stop_vent_1 := true;
             #Signal_Torche.Stop_vent_2 := true;
           #Start_algoritm_gaz_vozduh_1 := false;
           #Start_algoritm_gaz_vozduh_2 := false;
           IF #Frequency_1_State <> 0 THEN
             #Frequency_1_Cmd_off := 8;
           END_IF;

           IF #Frequency_2_State <> 0 THEN
             #Frequency_2_Cmd_off := 8;
           END_IF;

         END_IF;
    //**************************************************************************************************************     
         (*IF NOT Valve_Open THEN 
             ANY_Klapan_time := false;*)
         IF #After_alarm.Q = true THEN // если таймер прошел - переходим в режим 0
             #Signal_Torche.After_alarm_start := false;
           #Number_regim := 0;
           #Signal_Torche.Warning_bool_8 := true;
           #DO_Alarm := false;
           #Signal_Torche.Alarm_state := false;
           #Signal_Torche.After_stop_start := true; // запускаем Таймер после останова факела, для времени остывания факела и невыдачи в это время Warning
         END_IF;
         (*ELSIF (Valve_Open and (TEMP_TON_2_Q))  THEN

                   Warning := true;
                   ANY_Klapan_time := false;
                   IF  TEMP_TON_6_Q = true THEN
                     ANY_Time_after_alarms := false;
                     Rezerv_Alarmstop_on := false;
                     Number_regim := 0;
                     ANY_Stop_fakel := true; 
                   END_IF;

         END_IF;*)

     END_CASE;

     IF #Stop THEN // при нажатии кнопки Stop сбрасываем все таймеры, а так же запускаем запускаем Таймер после останова факела, для времени остывания факела и невыдачи в это время Warning

   //***********************************************// если версия прошивки 2 *************************************************************************************************            
         IF #Signal_Torche.Vers_number = 2 AND #Number_regim = 0 THEN
         #Frequency_1_Fail := 0; // сбарсываем ошибки приводов
         #Frequency_2_Fail := 0;
         #Frequency_1_Cmd_off := 8; // останавливаем привода
         #Frequency_2_Cmd_off := 8;
         #Signal_Torche.Stop_vent_1 := true; // останавливаем вентиляторы
         #Signal_Torche.Stop_vent_2 := true;
     END_IF;
     //********************************************************************** ************************************************************************************************        

       #Alarm_number := 0;
       #Signal_Torche.After_stop_start := true;
       #Signal_Torche.Sparking_start := false;
       #Signal_Torche.Spark_off_start := false;
       #Signal_Torche.Spark_on_start := FALSE;
       #Signal_Torche.After_alarm_start := false;
       #Signal_Torche.Stabilization_start:= false;
       #Signal_Torche.Venting_start:= false;

       #Spark_1_to_on := false;
       #Spark_2_to_on := false;
       #Spark_3_to_on := false;
       #Spark_4_to_on := false;
       (*#Signal_Torche.Warning_bool_8 := true;*)
       (*ANY_Klapan_time := true;*)
       #Signal_Torche.Privod_not_load := false;

       #DO_Alarm := false;
       #Signal_Torche.Alarm_state := false;
       #Valve_to_open := false;
       #Lamp_on_valve_open := false;

       #Number_regim := 0;

       (*
       #Signal_Torche.Time_after_alm_g := 60;
       #Signal_Torche.Time_stabiliz_g := 30;

       #Signal_Torche.Time_firing_g := 60;
       #Signal_Torche.Time_vent_g := 30;(**)

       #Signal_Torche.Time_stop_fire_g := 60;
       #Signal_Torche.Time_start_g := 55;
       #Signal_Torche.Time_klapan := 15;
       #Signal_Torche.Time_fire_off_g := 5;
       #Signal_Torche.Time_spark_off_g := 10;
       #Signal_Torche.Time_spark_on_g := 5;
       *)

       IF #Signal_Torche.Vers_number = 2 THEN
         IF #Frequency_1_Fail <> 0 THEN
             #Frequency_1_Cmd_Reset_Error := 8;
         END_IF;
         IF #Frequency_2_Fail <> 0 THEN
           #Frequency_2_Cmd_Reset_Error := 8;
         END_IF;
         #Start_algoritm_gaz_vozduh_1 := false;
         #Start_algoritm_gaz_vozduh_2 := false;
       END_IF;


     END_IF;
     //***********************************************Ручной режим работы факела *************************************             
   ELSIF #Man_fakel THEN //если в режиме ручной
       #Signal_Torche.Man_auto := true;
     (*IF Start THEN 
         Spark_1_to_on := true;
     ELSE
         Spark_1_to_on := false;
     END_IF;*)

       //***********************************************// если версия прошивки 2 **********************************************************************************************           
       IF #Signal_Torche.Vers_number = 2 THEN

           #Signal_Torche.Start_vent_1 := #Panel_vent_1_on; // возможность запуска вентиляторов с БАРКП 
           #Signal_Torche.Start_vent_2 := #Panel_vent_2_on;
           #Signal_Torche.Stop_vent_1 := #Panel_vent_1_off;
           #Signal_Torche.Stop_vent_2 := #Panel_vent_2_off;

           #Signal_Torche.Frequency_1_Mode := 4; // Режим работы приводов - ручной
           #Signal_Torche.Frequency_2_Mode := 4;
     END_IF;
     //*************************************************************************************************************** *********************************************************            
     IF #Valve_to_open_man THEN //***************** Возможность открытия клапана вручную****************
       #Valve_to_open := TRUE;
     ELSE
       #Valve_to_open := FALSE;
     END_IF;
   (*if Vers_number = 2 THEN
       IF Frequency_1_Fail <> 0 THEN
               Frequency_1_Cmd_Reset_Error := 4;
       END_IF;
       IF Frequency_2_Fail <> 0 THEN
               Frequency_2_Cmd_Reset_Error := 4;
       END_IF;
   END_IF;*)


   END_IF;

   IF #P_gaz_low THEN // индикация низкого давления газа
     #Lamp_P_zapal_low := true;
   ELSE
     #Lamp_P_zapal_low := false;
   END_IF;

   IF #Signal_Torche.Vers_number = 1 THEN // индикация горения факела
     #Lamp_1_on_door := #Temp_rozgik_FND_1;
     #Fire_is_off_1 := NOT #Temp_rozgik_FND_1;

   END_IF;
   //***********************************************// если версия прошивки 2 **************************************************************************************************** 
   IF #Signal_Torche.Vers_number = 2 THEN

     IF #Temp_rozgik_FND_1 AND #Temp_rozgik_FND_2 THEN // индикация горения факела
       #Lamp_1_on_door := true;
     END_IF;
     IF NOT #Temp_rozgik_FND_1 AND NOT #Temp_rozgik_FND_2 THEN
       #Lamp_1_on_door := false;
     END_IF;
     IF (NOT #Temp_rozgik_FND_1 AND #Temp_rozgik_FND_2) OR (#Temp_rozgik_FND_1 AND NOT #Temp_rozgik_FND_2) THEN
         #Lamp_1_on_door := #Signal_Torche.Fire_time_1;
     END_IF;


     IF #Temp_rozgik_FVD_1 AND #Temp_rozgik_FVD_2 THEN
       #Lamp_2_on_door := true;
     END_IF;
     IF NOT #Temp_rozgik_FVD_1 AND NOT #Temp_rozgik_FVD_2 THEN
       #Lamp_2_on_door := false;
     END_IF;
     IF (NOT #Temp_rozgik_FVD_1 AND #Temp_rozgik_FVD_2) OR (#Temp_rozgik_FVD_1 AND NOT #Temp_rozgik_FVD_2) THEN
         #Lamp_2_on_door := #Signal_Torche.Fire_time_1;
     END_IF;



     IF NOT (#Temp_rozgik_FND_1 AND #Temp_rozgik_FND_2) THEN
       #Fire_is_off_1 := true;
     ELSE
       #Fire_is_off_1 := false;
     END_IF;

     IF NOT (#Temp_rozgik_FVD_1 AND #Temp_rozgik_FVD_2) THEN
       #Fire_is_off_2 := true;
     ELSE
       #Fire_is_off_2 := false;
     END_IF;
   END_IF;

   //***************************************************************************************************************************************************************************
END_FUNCTION_BLOCK

FUNCTION "AI_Process" : Void   // FC1, FBD
{ S7_Optimized_Access := 'TRUE' }
VERSION : 0.1
BEGIN

REGION Network 1: Термопара на факеле
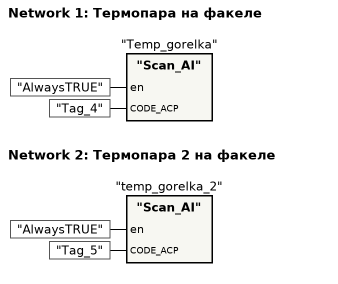
   IF "AlwaysTRUE" THEN
       "Temp_gorelka"(CODE_ACP := "Tag_4");   // "Scan_AI"
   END_IF;
END_REGION

REGION Network 2: Термопара 2 на факеле
   IF "AlwaysTRUE" THEN
       "temp_gorelka_2"(CODE_ACP := "Tag_5");   // "Scan_AI"
   END_IF;
END_REGION
END_FUNCTION

FUNCTION "Discrete_Process" : Void   // FC2, FBD
{ S7_Optimized_Access := 'TRUE' }
VERSION : 0.1
BEGIN

REGION Network 1: DI_16
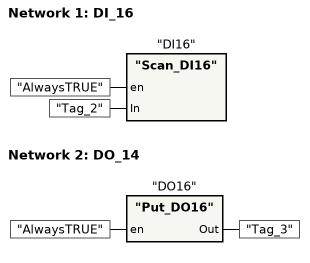
   IF "AlwaysTRUE" THEN
       "DI16"(In := "Tag_2");   // "Scan_DI16"
   END_IF;
END_REGION

REGION Network 2: DO_14
   IF "AlwaysTRUE" THEN
       "DO16"(Out => "Tag_3");   // "Put_DO16"
   END_IF;
END_REGION
END_FUNCTION

FUNCTION "Other" : Void   // FC3, SCL
{ S7_Optimized_Access := 'TRUE' }
VERSION : 0.1
BEGIN
   "test" := true;

   //***************Сведение команды старт/cтоп с верхнего уровня и команды с БРКП в единую команду****************************
   IF "MB_Start" OR "DI16".Slot.Pins[3] THEN
       "TP_start" := true;
   ELSIF NOT ("MB_Start" AND "DI16".Slot.Pins[3]) THEN
       "TP_start" := false;
   END_IF;

   IF "MB_Stop" OR "DI16".Slot.Pins[4] THEN
       "TP_stop" := true;
   ELSIF NOT ("MB_Stop" AND "DI16".Slot.Pins[4]) THEN
       "TP_stop" := false;
   END_IF;

   //***************Перекладывание для ВУ и БРКП**************
   //*******Сигнал Горит***************
   IF "Fire" THEN
       "DO16".Slot.Pins[0] := true;
   ELSIF NOT "Fire" THEN
       "DO16".Slot.Pins[0] := false;
   END_IF;

   //*******Идет подача искры***************
   IF "Spark_on" THEN
       "DO16".Slot.Pins[1] := true;
       "DO16".Slot.Pins[2] := true;
   ELSIF NOT "Spark_on" THEN
       "DO16".Slot.Pins[1] := false;
       "DO16".Slot.Pins[2] := true;
   END_IF;
END_FUNCTION

FUNCTION "Startup_parametrs" : Void   // FC4, SCL
{ S7_Optimized_Access := 'TRUE' }
VERSION : 0.1
BEGIN
   // Настройка аналоговых сигналов
   "Temp_gorelka".Signal_AI.VoltageInputType := false;
   "Temp_gorelka".Signal_AI.Scale_0_20mA := false;
   "Temp_gorelka".Signal_AI.H_Alarm_En := true;
   "Temp_gorelka".Signal_AI.HH_Alarm_En := true;
   "Temp_gorelka".Signal_AI.L_Alarm_En := false;
   "Temp_gorelka".Signal_AI.LL_Alarm_En := false;

   "temp_gorelka_2".Signal_AI.VoltageInputType := false;
   "temp_gorelka_2".Signal_AI.Scale_0_20mA := false;
   "temp_gorelka_2".Signal_AI.H_Alarm_En := true;
   "temp_gorelka_2".Signal_AI.HH_Alarm_En := true;
   "temp_gorelka_2".Signal_AI.L_Alarm_En := false;
   "temp_gorelka_2".Signal_AI.LL_Alarm_En := false;
   //************************************************Диапазон измерения датчика температуры**************************************
   "Temp_gorelka".Signal_AI.Scal_Max_Eu := 1100;
   "temp_gorelka_2".Signal_AI.Scal_Max_Eu := 1100;
   "Modbus_Buffer".Scal_max := 1100;
   "Temp_gorelka".Signal_AI.Scal_Min_Eu := -40;
   "temp_gorelka_2".Signal_AI.Scal_Min_Eu := -40;
   "Modbus_Buffer".Scal_min := -40;
   //************************************************Время зоны нечувствительности (защита от дребезга)**************************************
   "temp_gorelka_2".Signal_AI.HH_Delay := t#5s;
   "Temp_gorelka".Signal_AI.HH_Delay := t#5s;

   "DI16".Slot.Input_En := 16#FFFF;
   "DI16".Slot.Invert_En := 16#0000;
   "DO16".Slot.Output_En_out := 16#FFFF;
   "DO16".Slot.Invert_En := 16#0000;

   //..................................Факел................................
   "Torche_DB".Signal_Torche.Vers_number := 1; //номер версии прошивки факела
   "Torche_DB".Signal_Torche.Time_after_alm_g := 40;  //время после остановки факела до анализа температуры горения (сек)
   "Modbus_Buffer".Time_after_alarm := 40;
   "Torche_DB".Signal_Torche.Time_vent_g := 15;  //время вентиляции запальной трубы (сек)
   "Modbus_Buffer".Time_Venting := 15;
   "Torche_DB".Signal_Torche.Time_firing_g := 60;   //время розжига (сек)
   "Modbus_Buffer".Time_firing := 60;
   "Torche_DB".Signal_Torche.Time_spark_off_g := 10; // время отсутствия искры во время розжига (сек)
   "Modbus_Buffer".Time_spark_off := 10;
   "Torche_DB".Signal_Torche.Time_spark_on_g := 5; // время наличия искры во время розжига (сек)
   "Modbus_Buffer".Time_spark_on := 5;
   "Torche_DB".Signal_Torche.Time_stabiliz_g := 30; // время нстабилизации пламени (сек)
   "Modbus_Buffer".Time_stabil := 30;
   "Torche_DB".Signal_Torche.Time_stop_fire_g := 60; // время после аварийного останова до перехода в состояние готовность (сек)
   "Modbus_Buffer".Time_after_stop := 60;

   "Modbus_Buffer".Temp_curr_voltage := true; // Датчик температуры у нас - Voltage
   "Temp_gorelka".Signal_AI.VoltageInputType := true;
   "temp_gorelka_2".Signal_AI.VoltageInputType := true;
   "Modbus_Buffer".Temp_Fire := 150;
   "Temp_gorelka".Signal_AI.HH_Lim := 150;
   "temp_gorelka_2".Signal_AI.HH_Lim := 150;
   //..................................Modbus................................
   "MB_Parameters".MB_Load_req := true;
   "MB_Parameters".MP_Load_Port := "Local~CM1";
   "MB_Parameters".MB_Load_Baud := 9600;
   "MB_Parameters".MB_Load_Parity := 0;
   "MB_Parameters".MB_Addr := 1;



   //"DO_16_DB_07".Slot.Output_En_out := 16#FFFF;
   //"DO_CPU_DB".Slot.Output_En_out  := 16#FFFF;
   (*// Обе линии в учёте
   "DO_16_DB_07".Slot.Pins[6] := 0;
   "DO_16_DB_07".Slot.Pins[8] := 0;
   *)
   // Сюда надо добавить инициализацию пределов, уставок и флагов алярмов для всех AI, потом закоментировать
END_FUNCTION

ORGANIZATION_BLOCK "Main"   // OB1, LAD, ProgramCycle
TITLE = "Main Program Sweep (Cycle)"
{ S7_Optimized_Access := 'TRUE' }
VERSION : 0.1
   VAR_INPUT
      Initial_Call : Bool;   // Initial call of this OB
      Remanence : Bool;   // =True, if remanent data are available
   END_VAR
BEGIN

REGION Network 1: Обработка аналоговых сигналов
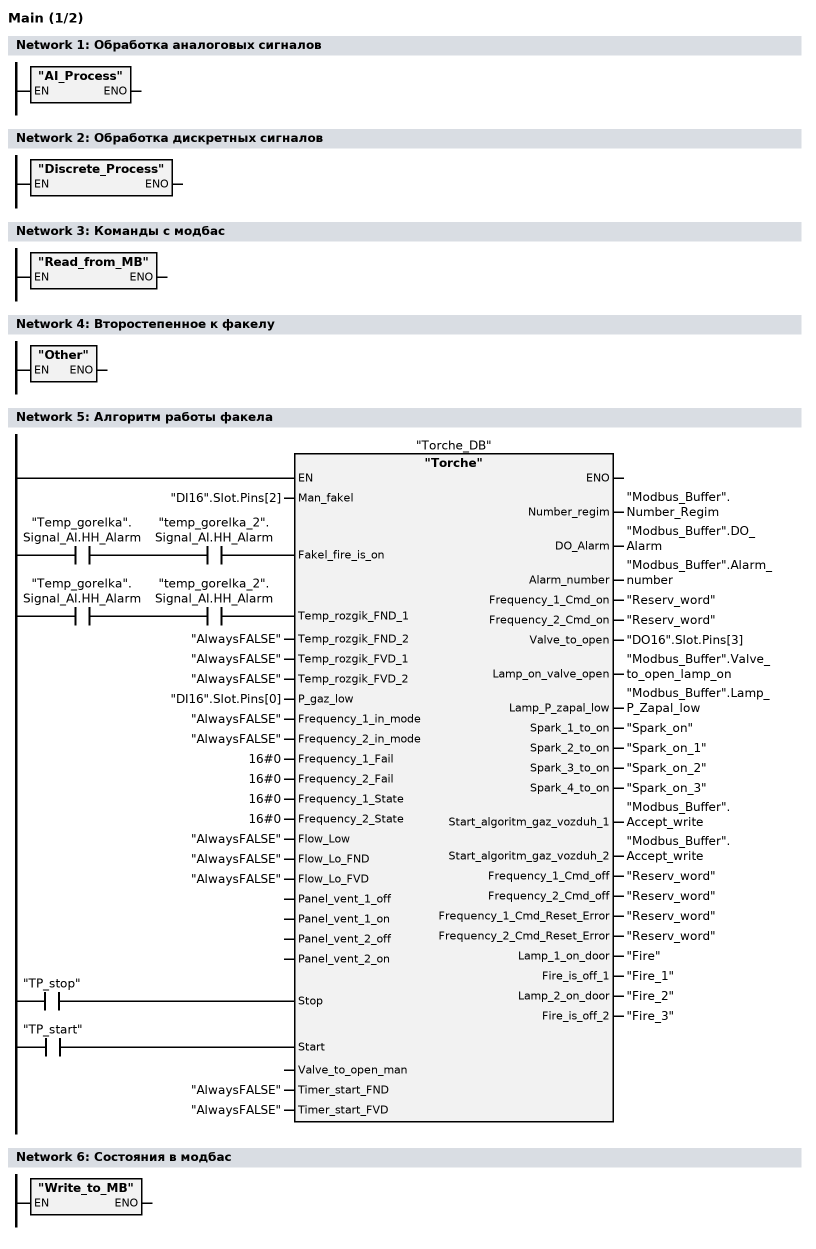
   RUNG wire#powerrail
      "AI_Process"()
   END_RUNG
   // the same network as SCL:
   "AI_Process"();
END_REGION

REGION Network 2: Обработка дискретных сигналов
   RUNG wire#powerrail
      "Discrete_Process"()
   END_RUNG
   // the same network as SCL:
   "Discrete_Process"();
END_REGION

REGION Network 3: Команды с модбас
   RUNG wire#powerrail
      "Read_from_MB"()
   END_RUNG
   // the same network as SCL:
   "Read_from_MB"();
END_REGION

REGION Network 4: Второстепенное к факелу
   RUNG wire#powerrail
      "Other"()
   END_RUNG
   // the same network as SCL:
   "Other"();
END_REGION

REGION Network 5: Алгоритм работы факела
   RUNG wire#powerrail
      "Torche_DB"(Fakel_fire_is_on := wire#w1, Temp_rozgik_FND_1 := wire#w2, Stop := wire#w3, Start := wire#w4, Man_fakel := "DI16".Slot.Pins[2], Temp_rozgik_FND_2 := "AlwaysFALSE", Temp_rozgik_FVD_1 := "AlwaysFALSE", Temp_rozgik_FVD_2 := "AlwaysFALSE", P_gaz_low := "DI16".Slot.Pins[0], Frequency_1_in_mode := "AlwaysFALSE", Frequency_2_in_mode := "AlwaysFALSE", Frequency_1_Fail := 16#0, Frequency_2_Fail := 16#0, Frequency_1_State := 16#0, Frequency_2_State := 16#0, Flow_Low := "AlwaysFALSE", Flow_Lo_FND := "AlwaysFALSE", Flow_Lo_FVD := "AlwaysFALSE", Panel_vent_1_off :=, Panel_vent_1_on :=, Panel_vent_2_off :=, Panel_vent_2_on :=, Valve_to_open_man :=, Timer_start_FND := "AlwaysFALSE", Timer_start_FVD := "AlwaysFALSE", Number_regim => "Modbus_Buffer".Number_Regim, DO_Alarm => "Modbus_Buffer".DO_Alarm, Alarm_number => "Modbus_Buffer".Alarm_number, Frequency_1_Cmd_on => "Reserv_word", Frequency_2_Cmd_on => "Reserv_word", Valve_to_open => "DO16".Slot.Pins[3], Lamp_on_valve_open => "Modbus_Buffer".Valve_to_open_lamp_on, Lamp_P_zapal_low => "Modbus_Buffer".Lamp_P_Zapal_low, Spark_1_to_on => "Spark_on", Spark_2_to_on => "Spark_on_1", Spark_3_to_on => "Spark_on_2", Spark_4_to_on => "Spark_on_3", Start_algoritm_gaz_vozduh_1 => "Modbus_Buffer".Accept_write, Start_algoritm_gaz_vozduh_2 => "Modbus_Buffer".Accept_write, Frequency_1_Cmd_off => "Reserv_word", Frequency_2_Cmd_off => "Reserv_word", Frequency_1_Cmd_Reset_Error => "Reserv_word", Frequency_2_Cmd_Reset_Error => "Reserv_word", Lamp_1_on_door => "Fire", Fire_is_off_1 => "Fire_1", Lamp_2_on_door => "Fire_2", Fire_is_off_2 => "Fire_3")
   END_RUNG
   RUNG wire#powerrail
      Contact( "Temp_gorelka".Signal_AI.HH_Alarm )
      Contact( "temp_gorelka_2".Signal_AI.HH_Alarm )
   END_RUNG wire#w1
   RUNG wire#powerrail
      Contact( "Temp_gorelka".Signal_AI.HH_Alarm )
      Contact( "temp_gorelka_2".Signal_AI.HH_Alarm )
   END_RUNG wire#w2
   RUNG wire#powerrail
      Contact( "TP_stop" )
   END_RUNG wire#w3
   RUNG wire#powerrail
      Contact( "TP_start" )
   END_RUNG wire#w4
   // the same network as SCL:
   "Torche_DB"(Man_fakel := "DI16".Slot.Pins[2],   // "Torche"
               Fakel_fire_is_on := "Temp_gorelka".Signal_AI.HH_Alarm AND "temp_gorelka_2".Signal_AI.HH_Alarm,
               Temp_rozgik_FND_1 := "Temp_gorelka".Signal_AI.HH_Alarm AND "temp_gorelka_2".Signal_AI.HH_Alarm,
               Temp_rozgik_FND_2 := "AlwaysFALSE",
               Temp_rozgik_FVD_1 := "AlwaysFALSE",
               Temp_rozgik_FVD_2 := "AlwaysFALSE",
               P_gaz_low := "DI16".Slot.Pins[0],
               Frequency_1_in_mode := "AlwaysFALSE",
               Frequency_2_in_mode := "AlwaysFALSE",
               Frequency_1_Fail := 16#0,
               Frequency_2_Fail := 16#0,
               Frequency_1_State := 16#0,
               Frequency_2_State := 16#0,
               Flow_Low := "AlwaysFALSE",
               Flow_Lo_FND := "AlwaysFALSE",
               Flow_Lo_FVD := "AlwaysFALSE",
               Stop := "TP_stop",
               Start := "TP_start",
               Timer_start_FND := "AlwaysFALSE",
               Timer_start_FVD := "AlwaysFALSE",
               Number_regim => "Modbus_Buffer".Number_Regim,
               DO_Alarm => "Modbus_Buffer".DO_Alarm,
               Alarm_number => "Modbus_Buffer".Alarm_number,
               Frequency_1_Cmd_on => "Reserv_word",
               Frequency_2_Cmd_on => "Reserv_word",
               Valve_to_open => "DO16".Slot.Pins[3],
               Lamp_on_valve_open => "Modbus_Buffer".Valve_to_open_lamp_on,
               Lamp_P_zapal_low => "Modbus_Buffer".Lamp_P_Zapal_low,
               Spark_1_to_on => "Spark_on",
               Spark_2_to_on => "Spark_on_1",
               Spark_3_to_on => "Spark_on_2",
               Spark_4_to_on => "Spark_on_3",
               Start_algoritm_gaz_vozduh_1 => "Modbus_Buffer".Accept_write,
               Start_algoritm_gaz_vozduh_2 => "Modbus_Buffer".Accept_write,
               Frequency_1_Cmd_off => "Reserv_word",
               Frequency_2_Cmd_off => "Reserv_word",
               Frequency_1_Cmd_Reset_Error => "Reserv_word",
               Frequency_2_Cmd_Reset_Error => "Reserv_word",
               Lamp_1_on_door => "Fire",
               Fire_is_off_1 => "Fire_1",
               Lamp_2_on_door => "Fire_2",
               Fire_is_off_2 => "Fire_3");
END_REGION

REGION Network 6: Состояния в модбас
   RUNG wire#powerrail
      "Write_to_MB"()
   END_RUNG
   // the same network as SCL:
   "Write_to_MB"();
END_REGION

REGION Network 7: Модбас RTU
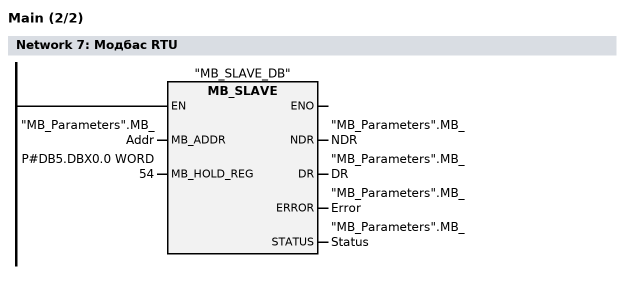
   "MB_SLAVE_DB"(MB_ADDR := "MB_Parameters".MB_Addr,   // MB_SLAVE
                 MB_HOLD_REG := P#DB5.DBX0.0 WORD 54,
                 NDR => "MB_Parameters".MB_NDR,
                 DR => "MB_Parameters".MB_DR,
                 ERROR => "MB_Parameters".MB_Error,
                 STATUS => "MB_Parameters".MB_Status);
END_REGION
END_ORGANIZATION_BLOCK

ORGANIZATION_BLOCK "Diagnostik"   // OB82, SCL, DiagnosticErrorInterrupt
{ S7_Optimized_Access := 'TRUE' }
VERSION : 0.1
   VAR_INPUT
      IO_State : Word;   // IO state of the HW object
      LADDR : Hw_Any;   // Hardware identifier
      Channel : UInt;   // Channel number
      MultiError : Bool;   // =true if more than one error is present
   END_VAR
BEGIN
END_ORGANIZATION_BLOCK

ORGANIZATION_BLOCK "Startup"   // OB100, FBD, Startup
TITLE = "Complete Restart"
{ S7_Optimized_Access := 'TRUE' }
VERSION : 0.1
   VAR_INPUT
      LostRetentive : Bool;   // True if retentive data are lost
      LostRTC : Bool;   // True if date and time are lost
   END_VAR
BEGIN

REGION Network 1: Вспомогательный блок
END_REGION

REGION Network 2: Установка параметров при запуске CPU
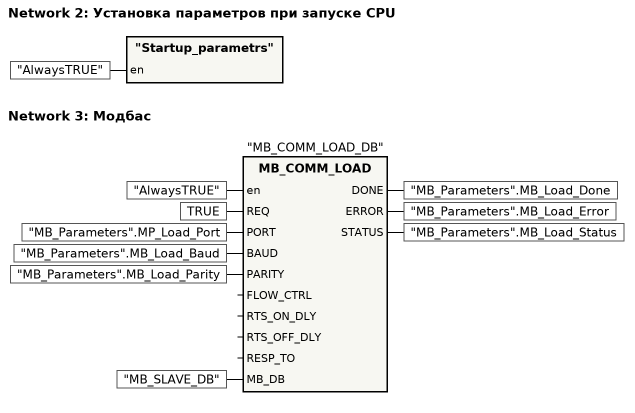
   IF "AlwaysTRUE" THEN "Startup_parametrs"(); END_IF;
END_REGION

REGION Network 3: Модбас
   IF "AlwaysTRUE" THEN
       "MB_COMM_LOAD_DB"(REQ := TRUE,   // MB_COMM_LOAD
                         PORT := "MB_Parameters".MP_Load_Port,
                         BAUD := "MB_Parameters".MB_Load_Baud,
                         PARITY := "MB_Parameters".MB_Load_Parity,
                         MB_DB := "MB_SLAVE_DB",
                         DONE => "MB_Parameters".MB_Load_Done,
                         ERROR => "MB_Parameters".MB_Load_Error,
                         STATUS => "MB_Parameters".MB_Load_Status);
   END_IF;
END_REGION
END_ORGANIZATION_BLOCK

// folder: Bits

FUNCTION "SetBitWord" : Void   // FC5, SCL
{ S7_Optimized_Access := 'TRUE' }
VERSION : 0.1
   VAR_INPUT
      pos : Int;
      value : Bool;
   END_VAR
   VAR_IN_OUT
      Data : Word;
   END_VAR
   VAR_TEMP
      mask : Word;
      v : Word;
   END_VAR
BEGIN

   IF #pos < 16 THEN
     #mask := 1;
     #mask := SHL(IN := #mask, N := #pos);
     IF #value THEN
       #Data := #Data OR #mask;
     ELSE
       #Data := #Data AND (NOT #mask);
     END_IF;
   END_IF;
END_FUNCTION

FUNCTION "GetBitWord" : Bool   // FC6, SCL
{ S7_Optimized_Access := 'TRUE' }
VERSION : 0.1
   VAR_INPUT
      Data : Word;
      pos : Int;
   END_VAR
   VAR_TEMP
      mask : Word;
      temp : Word;
   END_VAR
BEGIN

   #mask := 1;
   IF #pos < 16 THEN
     #mask := SHL(IN := #mask, N := #pos);
     #temp := #Data AND #mask;
     #GetBitWord := (#temp > 0);
   ELSE
     #GetBitWord := 0;
   END_IF;
END_FUNCTION

FUNCTION "GetBitByte" : Bool   // FC7, SCL
{ S7_Optimized_Access := 'TRUE' }
VERSION : 0.1
   VAR_INPUT
      Data : Byte;
      pos : Int;
   END_VAR
   VAR_TEMP
      mask : Byte;
      temp : Byte;
   END_VAR
BEGIN

   #mask := 1;
   IF #pos < 8 THEN
     #mask := SHL(IN := #mask, N := #pos);
     #temp := #Data AND #mask;
     #GetBitByte := (#temp > 0);
   ELSE
     #GetBitByte := 0;
   END_IF;
END_FUNCTION

// folder: Libs

FUNCTION_BLOCK "Scan_AI"   // FB1, SCL
TITLE = Analog input module block (current inputs)
{ S7_Optimized_Access := 'FALSE' }
NAME : Scan_AI
VERSION : 1.3
   VAR_INPUT
      CODE_ACP : Word := 0;   // Input ADC code
   END_VAR
   VAR
      Signal_AI : "dt_AI";
      HH_Timer : TON_TIME;
      H_Timer : TON_TIME;
      L_Timer : TON_TIME;
      LL_Timer : TON_TIME;
   END_VAR
   VAR_TEMP
      ACP_min : DInt;
      ACP_max : DInt;
      ACP_sc : DInt;   // Overload or shortcut code
      ACP_br : DInt;   // Negative overload or breakoff code
      Curr0_20_min : Real;
      Curr0_20_max : Real;
      Curr0_20_sc : Real;   // Overload or shortcut
      Curr0_20_br : Real;   // Negative overload or breakoff
      Curr4_20_min : Real;
      Curr4_20_max : Real;
      Curr4_20_sc : Real;   // Overload or shortcut
      Curr4_20_br : Real;   // Negative overload or breakoff TEMP
      Volt0_10_min : Real;
      Volt0_10_max : Real;
      Volt0_10_sc : Real;
      Temp_Real : Real;
      Temp_Int : Int;
      Temp_Start_Timer : Bool;
      Temp_Timer_State : Bool;
      temp_Min_Eu : Real;
      UEL : Byte;   // ВАУ
      UWL : Byte;   // ВПУ
      DWL : Byte;   // НПУ
      DEL : Byte;   // НАУ
      PNC : Byte;   // Параметр не контроллируется
      SIM : Byte;   // Симуляция
      MSK : Byte;   // Маскирование
      TST : Byte;   // Тестирование
   END_VAR
BEGIN

   // CONST
   //   ADC codes for Simatic S300
   //   Êîä ÀÖÏ     0-20  ìÀ    4-20  ìÀ     0-10 Â        Comment
   //    32512   |  23.52 ìÀ  | 22.81 ìÀ  |  11.759 Â  | Overload or shortcut
   //    27648   |  20.0  ìÀ  | 20.0  ìÀ  |  10.0 Â    | Normal
   //      1     |  723.4 íÀ  | 4.578 ìÀ  |  361.7 ìêÂ | Normal
   //      0     |    0.0 ìÀ  |   4   ìÀ  |  0.0 Â     | Normal
   //    -4865   |  -3.52 ìÀ  | 1.185 ìÀ  |  ----      | Negative overload or breakoff 
   #ACP_min := 0;
   #ACP_max := 27648;
   #ACP_sc := 32512;  // Overload or shortcut code
   #ACP_br := -4865;  // Negative overload or breakoff code (circuit only)
   #Curr0_20_min := 0.0;
   #Curr0_20_max := 20.0;
   #Curr0_20_sc := 23.52;  // Overload or shortcut
   #Curr0_20_br := -3.52;  // Negative overload or breakoff
   #Curr4_20_min := 4.0;
   #Curr4_20_max := 20.0;
   #Curr4_20_sc := 22.81;  // Overload or shortcut
   #Curr4_20_br := 1.185;  // Negative overload or breakoff
   #Volt0_10_min := 0.0;
   #Volt0_10_max := 10.0;
   #Volt0_10_sc := 11.759;

   #UEL := 2#00000001;
   #UWL := 2#00000010;
   #DWL := 2#00000100;
   #DEL := 2#00001000;
   #PNC := 2#00010000;
   #SIM := 2#00100000;
   #MSK := 2#01000000;
   #TST := 2#10000000;

   // 1) Îáÿçàòåëüíî ïîäàòü íà âõîä CODE_ACP çíà÷åíèå ñ ñîîòâåòñòâóþùåãî êàíàëà àíàëîãîâîãî ââîäà
   // 2) Îáÿçàòåëüíî âûñòàâèòü òèï ìàñøòàáèðîâàíèÿ Scale_Type, 1 ýòî 0-20 ìÀ à 0 ýòî 4-20 ìÀ 
   // 3) Îáÿçàòåëüíî âûñòàâèòü äèàïàçîíû ìàñøòàáèðîâàíèÿ Scal_Max_Eu è Scal_Min_Eu
   // 4) Âûñòàâèòü åñëè íåîáõîäèìî êîýôôèöèåíò ôèëüòðàöèè  K_filtr
   // 5) Ïðîâåðèòü ÷òî íå âêëþ÷åí ðåæèì ñèìóëÿöèè  Sim_En 


   //*   Ôîðìóëû ìàñøòàáèðîâàíèÿ:
   //*   Y = (X – Xmin ) * ( Ymax - Ymin ) / ( Xmax - Xmin ) + Ymin
   //*   X = (Y – Ymin ) * ( Xmax - Xmin ) / ( Ymax - Ymin ) + Xmin

   //------------------------------------------------------------------------
   //------------------Áëîê ðåæèìà ñèìóëÿöèè---------------------------------
   //------------------------------------------------------------------------ 

   //Åñëè ðåæèì ñèìóëÿöèè âêëþ÷åí òî èñïîëüçóåì çíà÷åíèå Sim_Value
   IF #Signal_AI.Sim_En THEN
       // Ìàñøòàáèðóåì çíà÷åíèå ñèìóëÿöèè â êîä ÀÖÏ - íå èñïîëüçóåòñÿ, òàê êàê èç-çà ðàçíûõ ðåæèìîâ 
       //  (òîê 4-20/0-20, íàïðÿæåíèå) ñëîæíî îäíîçíà÷íî ñäåëàòü ïðåîáðàçîâàíèå â ñîîòâåòñòâóþùóþ âåëèöèíó ÀÖÏ
       //#Signal_AI.Acp := ROUND (( #Signal_AI.Sim_Value - #Signal_AI.Scal_Min_Eu)*DINT_TO_REAL(#ACP_max - #ACP_min) /
       //                         ( #Signal_AI.Scal_Max_Eu - #Signal_AI.Scal_Min_Eu) + DINT_TO_REAL(#ACP_min));
       #Signal_AI.State := #Signal_AI.State OR #SIM;
       #Temp_Real := #Signal_AI.Sim_Value;
   ELSE
       // èíà÷å èñïîëüçóåì àíàëîãîâûé âõîä
       #Signal_AI.State := #Signal_AI.State AND (NOT(#SIM));
       #Signal_AI.Acp := WORD_TO_INT(#CODE_ACP);

       //------------------------------------------------------------------------
       //-------------Áëîê ìàñøòàáèðîâàíèÿ---------------------------------------
       //------------------------------------------------------------------------
       IF #Signal_AI.VoltageInputType THEN
           // âõîä íàïðÿæåíèÿ
           // îïðåäåëåíèå íàïðÿæåíèÿ èç êîäà àöï  
           #Signal_AI.Voltage := DINT_TO_REAL(#Signal_AI.Acp - #ACP_min) * (#Volt0_10_max - #Volt0_10_min) / (DINT_TO_REAL(#ACP_max - #ACP_min)) + #Volt0_10_min;
           // îïðåäåëèì ýêâèâàëåíò òîêà ÷åðåç âõîäíîå ñîïðîòèâëåíèå
           IF #Signal_AI.Resistance > 0 THEN
               #Signal_AI.Circuit := #Signal_AI.Voltage / #Signal_AI.Resistance;
               // îïðåäåëåíèå çíà÷åíèÿ ñèãíàëà â èíæ. âåëè÷èíå èç ýêâèâàëåíòà òîêà 
               IF #Signal_AI.Scale_0_20mA THEN
                   #Temp_Real := (#Signal_AI.Circuit - #Curr0_20_min) * (#Signal_AI.Scal_Max_Eu - #Signal_AI.Scal_Min_Eu) / (#Curr0_20_max - #Curr0_20_min) + #Signal_AI.Scal_Min_Eu;
               ELSE
                   #Temp_Real := (#Signal_AI.Circuit - #Curr4_20_min) * (#Signal_AI.Scal_Max_Eu - #Signal_AI.Scal_Min_Eu) / (#Curr4_20_max - #Curr4_20_min) + #Signal_AI.Scal_Min_Eu;
               END_IF;
           ELSE
               // îïðåäåëåíèå çíà÷åíèÿ ñèãíàëà â èíæ. âåëè÷èíå èç êîäà àöï 
               #Temp_Real := DINT_TO_REAL(#Signal_AI.Acp - #ACP_min) * (#Signal_AI.Scal_Max_Eu - #Signal_AI.Scal_Min_Eu) / (DINT_TO_REAL(#ACP_max - #ACP_min)) + #Signal_AI.Scal_Min_Eu;
           END_IF;

       ELSE
           // òîêîâûé âõîä
           IF #Signal_AI.Scale_0_20mA THEN          // Åñëè òèï ìàñøòàáèðîâàíèÿ 0-20 ìÀ òî
               // îïðåäåëåíèå òîêà èç êîäà àöï 
               #Signal_AI.Circuit := DINT_TO_REAL(#Signal_AI.Acp - #ACP_min) * (#Curr0_20_max - #Curr0_20_min) / (DINT_TO_REAL(#ACP_max - #ACP_min)) + #Curr0_20_min;
           ELSE                                    // Èíà÷å åñëè òèï ìàñøòàáèðîâàíèÿ 4-20 ìÀ òî
               // îïðåäåëåíèå òîêà èç êîäà àöï  
               #Signal_AI.Circuit := DINT_TO_REAL(#Signal_AI.Acp - #ACP_min) * (#Curr4_20_max - #Curr4_20_min) / (DINT_TO_REAL(#ACP_max - #ACP_min)) + #Curr4_20_min;
           END_IF;

           // îïðåäåëåíèå çíà÷åíèÿ ñèãíàëà â èíæ. âåëè÷èíå èç êîäà àöï
           IF (#Signal_AI.Scale_0_20mA AND #Signal_AI.Input_4mA_on_0_20mA) THEN// Åñëè äàò÷èê 4-20ìÀ èñïîëüçóåòñÿ íà âõîäå 0-20ìÀ
               // ñäâèãàåì âíèç íà 25% íèæíèé ïðåäåë äàò÷èêà, äî 0ìÀ 
               #temp_Min_Eu := #Signal_AI.Scal_Min_Eu - ((#Signal_AI.Scal_Max_Eu - #Signal_AI.Scal_Min_Eu) / 4.0);
               #Temp_Real := DINT_TO_REAL(#Signal_AI.Acp - #ACP_min) * (#Signal_AI.Scal_Max_Eu - #temp_Min_Eu) / (DINT_TO_REAL(#ACP_max - #ACP_min)) + #temp_Min_Eu;
           ELSE
               #Temp_Real := DINT_TO_REAL(#Signal_AI.Acp - #ACP_min) * (#Signal_AI.Scal_Max_Eu - #Signal_AI.Scal_Min_Eu) / (DINT_TO_REAL(#ACP_max - #ACP_min)) + #Signal_AI.Scal_Min_Eu;
           END_IF;
       END_IF;


   END_IF;

   //------------------------------------------------------------------------
   //-----------Áëîê ôèëüòðàöèè (ñãëàæèâàíèÿ) àíàëîãîâîãî ñèãíàëà------------
   // Åñëè ðåæèì ôèëüòðàöèè âêëþ÷åí ðàñ÷èòàòü çíà÷åíèå ïî ôîðìóëå Óâûõ=Óïîñë + Êôèëòð*( Óòåê - Óïîñë)
   // ïðè ñãëàæèâàíèè ïî íèæåïðèâåäåííîé  ôîðìóëå ïðîèñõîäèò ïîñêàíîâîå ïðèáëèæåíèå âûõîäíîãî
   // çíà÷åíèÿ ê òåêóùåìó (ðåàëüíîìó) ñèãíàëó
   //------------------------------------------------------------------------

   IF #Signal_AI.K_filtr > 0 THEN
       #Signal_AI.Value := #Signal_AI.Value_LastScan + #Signal_AI.K_filtr * (#Temp_Real - #Signal_AI.Value_LastScan);
       //Çàïîìèíàåì òåêóùåå çíà÷åíèå êàê çíà÷åíèå ñ ïîñëåäíåãî ñêàíà
       #Signal_AI.Value_LastScan := #Signal_AI.Value;
   ELSE
       // âûñòàâëÿåì òåêóùåå çíà÷åíèå 
       #Signal_AI.Value := #Temp_Real;
   END_IF;

   //------------------------------------------------------------------------
   //Áëîê ïðîâåðêè âûõîäà çíà÷åíèÿ ñèãíàëà èç ðàáî÷åãî äèàïàçîíà-------------
   //------------------------------------------------------------------------

   IF #Signal_AI.Value > #Signal_AI.Scal_Max_Eu THEN      //Ïðè âûõîäå çíà÷åíèÿ ñèãíàëà èç çàäàííîãî äèàïàçîíà ïðèðàâíèâàåì åãî ê âåðõíåìó ïðåäåëó ýòîãî äèàïàçîíà
       #Signal_AI.Value := #Signal_AI.Scal_Max_Eu;
       #Signal_AI.Scal_Max_Upper := true;                 //çàæèãàåì ôëàã ïðåâûøåíèÿ çíà÷åíèÿ ñèãíàëà âåðõíåãî ïðåäåëà äèàïàçîíà ìàñøòàáèðîâàíèÿ
   ELSE
       #Signal_AI.Scal_Max_Upper := false;
   END_IF;

   IF #Signal_AI.Value < #Signal_AI.Scal_Min_Eu THEN      //Ïðè âûõîäå çíà÷åíèÿ ñèãíàëà èç çàäàííîãî äèàïàçîíà ïðèðàâíèâàåì åãî ê íèæíåìó ïðåäåëó  ýòîãî äèàïàçîíà
       #Signal_AI.Value := #Signal_AI.Scal_Min_Eu;
       #Signal_AI.Scal_Min_Under := true;                 //çàæèãàåì ôëàã  çíà÷åíèÿ ñèãíàëà íèæå íèæíåãî ïðåäåëà äèàïàçîíà ìàñøòàáèðîâàíèÿ
   ELSE
       #Signal_AI.Scal_Min_Under := false;
   END_IF;

   //------------------------------------------------------------------------
   //---------Áëîê ïðîâåðêè ïðåâûøåíèÿ óñòàâêè ïî âåðõíåìó àâàðèéíîìó ïðåäåëó
   //------------------------------------------------------------------------
   IF #Signal_AI.HH_Alarm THEN    // Åñëè åñòü àâàðèÿ òî äëÿ îáåñïå÷åíèÿ ãèñòåðåçèñà 
       // Ðàçðåøåíèå íà ñòàðò òàéìåðà åñëè ïðîâåðêà ðàçðåøåíà è çíà÷åíèå ïðåâûøàåò óñòàâêó
       #Temp_Start_Timer := #Signal_AI.HH_Alarm_En AND (#Signal_AI.Value > (#Signal_AI.HH_Lim - #Signal_AI.HH_DeadBand));
   ELSE
       // Ðàçðåøåíèå íà ñòàðò òàéìåðà åñëè ïðîâåðêà ðàçðåøåíà è çíà÷åíèå ïðåâûøàåò óñòàâêó
       #Temp_Start_Timer := #Signal_AI.HH_Alarm_En AND (#Signal_AI.Value > (#Signal_AI.HH_Lim + #Signal_AI.HH_DeadBand));
   END_IF;

   #HH_Timer(IN := #Temp_Start_Timer // IN: BOOL
             ,
             PT := #Signal_AI.HH_Delay // IN: TIME
   );

   //åñëè  âðåìÿ çàäåðæêè èñòåêëî òî çàæèãàåì ôëàã àâàðèè , èíà÷å ãàñèì åãî
   IF #HH_Timer.Q THEN
       #Signal_AI.HH_Alarm := true;
       #Signal_AI.State := #Signal_AI.State OR #UEL;
   ELSE
       #Signal_AI.HH_Alarm := false;
       #Signal_AI.State := #Signal_AI.State AND (NOT(#UEL));
   END_IF;

   //------------------------------------------------------------------------
   //Áëîê ïðîâåðêè ïðåâûøåíèÿ óñòàâêè ïî âåðõíåìó ïðåäóïðåäèòåëüíîìó ïðåäåëó
   //------------------------------------------------------------------------
   IF #Signal_AI.H_Alarm THEN    // Åñëè åñòü àâàðèÿ òî äëÿ îáåñïå÷åíèÿ ãèñòåðåçèñà 
       // Ðàçðåøåíèå íà ñòàðò òàéìåðà åñëè ïðîâåðêà ðàçðåøåíà è çíà÷åíèå ïðåâûøàåò óñòàâêó
       #Temp_Start_Timer := #Signal_AI.H_Alarm_En AND (#Signal_AI.Value > (#Signal_AI.H_Lim - #Signal_AI.H_DeadBand));
   ELSE
       // Ðàçðåøåíèå íà ñòàðò òàéìåðà åñëè ïðîâåðêà ðàçðåøåíà è çíà÷åíèå ïðåâûøàåò óñòàâêó
       #Temp_Start_Timer := #Signal_AI.H_Alarm_En AND (#Signal_AI.Value > (#Signal_AI.H_Lim + #Signal_AI.H_DeadBand));
   END_IF;

   #H_Timer(IN := #Temp_Start_Timer // IN: BOOL
            ,
            PT := #Signal_AI.H_Delay // IN: TIME
   );

   //åñëè  âðåìÿ çàäåðæêè èñòåêëî òî çàæèãàåì ôëàã àâàðèè , èíà÷å ãàñèì åãî
   IF #H_Timer.Q THEN
       #Signal_AI.H_Alarm := true;
       #Signal_AI.State := #Signal_AI.State OR #UWL;
   ELSE
       #Signal_AI.H_Alarm := false;
       #Signal_AI.State := #Signal_AI.State AND (NOT(#UWL));
   END_IF;

   //------------------------------------------------------------------------
   //--Áëîê ïðîâåðêè ïðåâûøåíèÿ óñòàâêè ïî íèæíåìó ïðåäóïðåäèòåëüíîìó ïðåäåëó
   //------------------------------------------------------------------------
   IF #Signal_AI.L_Alarm THEN    // Åñëè åñòü àâàðèÿ òî äëÿ îáåñïå÷åíèÿ ãèñòåðåçèñà 
       #Temp_Start_Timer := #Signal_AI.L_Alarm_En AND (#Signal_AI.Value < (#Signal_AI.L_Lim + #Signal_AI.L_DeadBand));   // Ðàçðåøåíèå íà ñòàðò òàéìåðà åñëè ïðîâåðêà ðàçðåøåíà è çíà÷åíèå ïðåâûøàåò óñòàâêó
   ELSE
       #Temp_Start_Timer := #Signal_AI.L_Alarm_En AND (#Signal_AI.Value < (#Signal_AI.L_Lim - #Signal_AI.L_DeadBand));   // Ðàçðåøåíèå íà ñòàðò òàéìåðà åñëè ïðîâåðêà ðàçðåøåíà è çíà÷åíèå ïðåâûøàåò óñòàâêó
   END_IF;

   #L_Timer(IN := #Temp_Start_Timer // IN: BOOL
            ,
            PT := #Signal_AI.L_Delay // IN: TIME
   );

   //åñëè  âðåìÿ çàäåðæêè èñòåêëî òî çàæèãàåì ôëàã àâàðèè , èíà÷å ãàñèì åãî
   IF #L_Timer.Q THEN
       #Signal_AI.L_Alarm := true;
       #Signal_AI.State := #Signal_AI.State OR #DWL;
   ELSE
       #Signal_AI.L_Alarm := false;
       #Signal_AI.State := #Signal_AI.State AND (NOT(#DWL));
   END_IF;

   //------------------------------------------------------------------------
   //-------Áëîê ïðîâåðêè ïðåâûøåíèÿ óñòàâêè ïî íèæíåìó àâàðèéíîìó ïðåäåëó---
   //------------------------------------------------------------------------
   IF #Signal_AI.LL_Alarm THEN    // Åñëè åñòü àâàðèÿ òî äëÿ îáåñïå÷åíèÿ ãèñòåðåçèñà 
       #Temp_Start_Timer := #Signal_AI.LL_Alarm_En AND (#Signal_AI.Value < (#Signal_AI.LL_Lim + #Signal_AI.LL_DeadBand));   // Ðàçðåøåíèå íà ñòàðò òàéìåðà åñëè ïðîâåðêà ðàçðåøåíà è çíà÷åíèå ïðåâûøàåò óñòàâêó
   ELSE
       #Temp_Start_Timer := #Signal_AI.LL_Alarm_En AND (#Signal_AI.Value < (#Signal_AI.LL_Lim - #Signal_AI.LL_DeadBand));   // Ðàçðåøåíèå íà ñòàðò òàéìåðà åñëè ïðîâåðêà ðàçðåøåíà è çíà÷åíèå ïðåâûøàåò óñòàâêó
   END_IF;

   #LL_Timer(IN := #Temp_Start_Timer // IN: BOOL
             ,
             PT := #Signal_AI.LL_Delay // IN: TIME
   );

   //åñëè  âðåìÿ çàäåðæêè èñòåêëî òî çàæèãàåì ôëàã àâàðèè , èíà÷å ãàñèì åãî
   IF #LL_Timer.Q THEN
       #Signal_AI.LL_Alarm := true;
       #Signal_AI.State := #Signal_AI.State OR #DEL;
   ELSE
       #Signal_AI.LL_Alarm := false;
       #Signal_AI.State := #Signal_AI.State AND (NOT(#DEL));
   END_IF;

   //Определяем состояние маскирования
   IF (#Signal_AI.HH_Alarm_En AND #Signal_AI.H_Alarm_En AND #Signal_AI.L_Alarm_En AND #Signal_AI.LL_Alarm_En) THEN
       #Signal_AI.State := #Signal_AI.State AND (NOT (#MSK));// OR #MSK;
   ELSE
       #Signal_AI.State := #Signal_AI.State OR #MSK;// AND (NOT (#MSK));
   END_IF;


   //------------------------------------------------------------------------
   //------Áëîê ïðîâåðêè íà êîðîòêîå çàìûêàíèå è îáðûâ-----------------------
   //------------------------------------------------------------------------
   IF (NOT #Signal_AI.Sim_En) THEN
       // Ïðîâåðêà íà êîðîòêîå çàìûêàíèå.
       #Signal_AI.Short_Circuit := (#Signal_AI.Acp >= #ACP_sc);

       // Ïðîâåðêà íà îáðûâ.
       IF #Signal_AI.VoltageInputType AND (#Signal_AI.Resistance > 0) THEN
           // âõîä íàïðÿæåíèÿ ñ ïðåîáðàçîâàíèåì â òîêîâûé
           IF #Signal_AI.Scale_0_20mA THEN
               #Signal_AI.Break := (#Signal_AI.Circuit <= #Curr0_20_br);
           ELSE
               #Signal_AI.Break := (#Signal_AI.Circuit <= #Curr4_20_br);
           END_IF;
       ELSE
           // òîêîâûé âõîä
           IF (#Signal_AI.Scale_0_20mA AND #Signal_AI.Input_4mA_on_0_20mA) THEN
               #Signal_AI.Break := (#Signal_AI.Circuit <= #Curr4_20_br);
           ELSE
               #Signal_AI.Break := (#Signal_AI.Acp <= #ACP_br);
           END_IF;
       END_IF;


       //  Ïðè îáðûâå èëè êîðîòêîì çàìûêàíèè  ãàñèì ôëàãè ñðàáàòûâàíèÿ óñòàâîê
       IF (#Signal_AI.Short_Circuit OR #Signal_AI.Break) THEN
           #Signal_AI.HH_Alarm := false;
           #Signal_AI.H_Alarm := false;
           #Signal_AI.L_Alarm := false;
           #Signal_AI.LL_Alarm := false;
           #Signal_AI.Chan_Fail := true;
           #Signal_AI.State := #Signal_AI.State OR #PNC;
       ELSE
           #Signal_AI.Chan_Fail := false;
           #Signal_AI.State := #Signal_AI.State AND (NOT(#PNC));
       END_IF;

   ELSE
       #Signal_AI.Short_Circuit := false;
       #Signal_AI.Break := false;
       #Signal_AI.Chan_Fail := false;
   END_IF;

   // Режим маскирования (или тестирования ?) - ХЗ. сделал как-будто это одно и то же
   IF (#Signal_AI.Mask_mode) THEN
       #Signal_AI.HH_Alarm_Logic := false;
       #Signal_AI.H_Alarm_Logic := false;
       #Signal_AI.L_Alarm_Logic := false;
       #Signal_AI.LL_Alarm_Logic := false;
       #Signal_AI.Chan_Fail_Logic := false;
       #Signal_AI.Test_mode := true;
   ELSE
       #Signal_AI.HH_Alarm_Logic := #Signal_AI.HH_Alarm;
       #Signal_AI.H_Alarm_Logic := #Signal_AI.H_Alarm;
       #Signal_AI.L_Alarm_Logic := #Signal_AI.L_Alarm;
       #Signal_AI.LL_Alarm_Logic := #Signal_AI.LL_Alarm;
       #Signal_AI.Chan_Fail_Logic := #Signal_AI.Chan_Fail;
       #Signal_AI.Test_mode := false;
   END_IF;

   // Квитирование аварий по аналоговым параметрам (моргание на HMI)
   IF ((#Signal_AI.HH_Alarm AND NOT #Signal_AI.Ack_HH) OR (#Signal_AI.LL_Alarm AND NOT #Signal_AI.Ack_LL)) THEN
       #Signal_AI.Ack_Alarm := 1;
   ELSIF ((#Signal_AI.HH_Alarm AND #Signal_AI.Ack_HH) OR (#Signal_AI.LL_Alarm AND #Signal_AI.Ack_LL)) THEN
       #Signal_AI.Ack_Alarm := 2;
   ELSIF (NOT #Signal_AI.HH_Alarm AND NOT #Signal_AI.LL_Alarm) THEN
       #Signal_AI.Ack_Alarm := 0;
       #Signal_AI.Ack_HH := false;
       #Signal_AI.Ack_LL := false;
   END_IF;

   IF ((#Signal_AI.H_Alarm AND NOT #Signal_AI.Ack_H) OR (#Signal_AI.L_Alarm AND NOT #Signal_AI.Ack_L)) THEN
       #Signal_AI.Ack_Warning := 1;
   ELSIF ((#Signal_AI.H_Alarm AND #Signal_AI.Ack_H) OR (#Signal_AI.L_Alarm AND #Signal_AI.Ack_L)) THEN
       #Signal_AI.Ack_Warning := 2;
   ELSIF (NOT #Signal_AI.H_Alarm AND NOT #Signal_AI.L_Alarm) THEN
       #Signal_AI.Ack_Warning := 0;
       #Signal_AI.Ack_H := false;
       #Signal_AI.Ack_L := false;
   END_IF;

   // Закраска прямоугольников на HMI
   IF (#Signal_AI.Mask_mode) THEN
       #Signal_AI.State_color := 3;
   ELSIF (#Signal_AI.Chan_Fail) THEN
       #Signal_AI.State_color := 4;
   ELSIF (#Signal_AI.HH_Alarm OR #Signal_AI.LL_Alarm) THEN
       #Signal_AI.State_color := 2;
   ELSIF (#Signal_AI.H_Alarm OR #Signal_AI.L_Alarm) THEN
       #Signal_AI.State_color := 1;
   ELSE
       #Signal_AI.State_color := 0;
   END_IF;
END_FUNCTION_BLOCK

FUNCTION_BLOCK "Scan_DI32"   // FB2, SCL
TITLE = '32-bit DI module scan'
{ S7_Optimized_Access := 'FALSE' }
NAME : ScanDI32
VERSION : 1.2
   VAR_INPUT
      In : DWord;
   END_VAR
   VAR
      Slot : Struct
         Input_En : DWord;   // enable input mask
         Filter_En : DWord;   // filter mask
         Invert_En : DWord;   // invert mask
         Sim_En : DWord;   // simulate enable mask
         Sim_Value : DWord;   // simulate value
         Input : DWord;   // In after inverting
         Value : DWord;   // Result after enable and filtering
         Value_Last_Scan : DWord;   // intermediate value
         Pins : Array[0..31] of Bool;   // hardware pins (accordance byte order)
      END_STRUCT;
   END_VAR
   VAR_TEMP
      Temp : DWord;
      Temp_In : DWord;
      i : Int;
      Hi : Word;
      Lo : Word;
   END_VAR
BEGIN




   #Temp_In := #In;
   #Slot.Input := #Temp_In XOR #Slot.Invert_En;         // Инвертирование сигналов 
   #Temp_In := #Slot.Input AND #Slot.Input_En;       // Проходят  только разрешенные синалы     
   #Temp := #Slot.Value_Last_Scan XOR #Temp_In;   // Выделение битов изменившихся за период таймаута
   #Temp := #Temp AND #Slot.Filter_En;            // Проверяем наличие разрешения на фильтрование от дребезга
   #Slot.Value := #Slot.Value AND #Temp;                // Сохраняем биты которые не должны изменится и обнуляем все остальные
   #Temp := NOT #Temp;                           // Инвертируем
   #Temp := #Temp AND #Temp_In;                   // Изменившиеся биты обнуляеми а не изменившиеся с последнего скана биты запоминаем 
   #Slot.Value := #Slot.Value OR #Temp;                 // Формируем выход 
   #Slot.Value_Last_Scan := #Temp_In;                   // Запоминаем текущее значение как значение последнего скана

   // При включенной симуляции заменяем исходное значение на Sim_Value
   #Slot.Value := (#Slot.Sim_En AND #Slot.Sim_Value) OR ((NOT #Slot.Sim_En) AND #Slot.Value);

   #Hi := DWORD_TO_WORD(SHR(IN := #Slot.Value, N := 16));
   #Lo := DWORD_TO_WORD(#Slot.Value);
   FOR #i := 0 TO 7 DO
     #Slot.Pins[#i + 24] := "GetBitWord"(Data := #Lo,
                                         pos := #i);
     #Slot.Pins[#i + 16] := "GetBitWord"(Data := #Lo,
                                         pos := #i + 8);
     #Slot.Pins[#i + 8] := "GetBitWord"(Data := #Hi,
                                        pos := #i);
     #Slot.Pins[#i] := "GetBitWord"(Data := #Hi,
                                    pos := #i + 8);
   END_FOR;
END_FUNCTION_BLOCK

FUNCTION_BLOCK "Scan_DI16"   // FB3, SCL
TITLE = '16-bit DI module scan'
{ S7_Optimized_Access := 'FALSE' }
NAME : ScanDI16
VERSION : 1.2
   VAR_INPUT
      In : Word;
   END_VAR
   VAR
      Slot : Struct
         Input_En : Word;   // enable input mask
         Filter_En : Word;   // filter mask
         Invert_En : Word;   // invert mask
         Sim_En : Word;   // simulate enable mask
         Sim_Value : Word;   // simulate value
         Input : Word;   // In after inverting
         Value : Word;   // Result after enable and filtering
         Value_Last_Scan : Word;   // intermediate value
         Pins : Array[0..15] of Bool;   // hardware pins (accordance byte order)
      END_STRUCT;
   END_VAR
   VAR_TEMP
      Temp : Word;
      Temp_In : Word;
      i : Int;
   END_VAR
BEGIN




   #Temp_In := #In;
   #Slot.Input := #Temp_In XOR #Slot.Invert_En;         // Инвертирование сигналов 
   #Temp_In := #Slot.Input AND #Slot.Input_En;      // Проходят  только разрешенные синалы     
   #Temp := #Slot.Value_Last_Scan XOR #Temp_In;   // Выделение битов изменившихся за период таймаута
   #Temp := #Temp AND #Slot.Filter_En;            // Проверяем наличие разрешения на фильтрование от дребезга
   #Slot.Value := #Slot.Value AND #Temp;                // Сохраняем биты которые не должны изменится и обнуляем все остальные
   #Temp := NOT #Temp;                           // Инвертируем
   #Temp := #Temp AND #Temp_In;                  // Изменившиеся биты обнуляеми а не изменившиеся с последнего скана биты запоминаем 
   #Slot.Value := #Slot.Value OR #Temp;                 // Формируем выход 
   #Slot.Value_Last_Scan := #Temp_In;                   // Запоминаем текущее значение как значение последнего скана

   // При включенной симуляции заменяем исходное значение на Sim_Value
   #Slot.Value := (#Slot.Sim_En AND #Slot.Sim_Value) OR ((NOT #Slot.Sim_En) AND #Slot.Value);

   FOR #i := 0 TO 7 DO
     #Slot.Pins[#i + 8] := "GetBitWord"(Data := #Slot.Value,
                                        pos := #i);
     #Slot.Pins[#i] := "GetBitWord"(Data := #Slot.Value,
                                    pos := #i + 8);
   END_FOR;
END_FUNCTION_BLOCK

FUNCTION_BLOCK "Scan_DI08"   // FB4, SCL
TITLE = '8-bit DI module scan'
{ S7_Optimized_Access := 'FALSE' }
NAME : ScanDI08
VERSION : 1.2
   VAR_INPUT
      In : Byte;
   END_VAR
   VAR
      Slot : Struct
         Input_En : Byte;   // enable input mask
         Filter_En : Byte;   // filter mask
         Invert_En : Byte;   // invert mask
         Sim_En : Byte;   // simulate enable mask
         Sim_Value : Byte;   // simulate value
         Input : Byte;   // In after inverting
         Value : Byte;   // Result after enable and filtering
         Value_Last_Scan : Byte;   // intermediate value
         Pins : Array[0..7] of Bool;   // hardware pins (accordance byte order)
      END_STRUCT;
   END_VAR
   VAR_TEMP
      Temp : Byte;
      Temp_In : Byte;
      i : Int;
   END_VAR
BEGIN




   #Temp_In := #In;
   #Slot.Input := #Temp_In XOR #Slot.Invert_En;         // Инвертирование сигналов 
   #Temp_In := #Slot.Input AND #Slot.Input_En;      // Проходят  только разрешенные синалы     
   #Temp := #Slot.Value_Last_Scan XOR #Temp_In;   // Выделение битов изменившихся за период таймаута
   #Temp := #Temp AND #Slot.Filter_En;            // Проверяем наличие разрешения на фильтрование от дребезга
   #Slot.Value := #Slot.Value AND #Temp;                // Сохраняем биты которые не должны изменится и обнуляем все остальные
   #Temp := NOT #Temp;                           // Инвертируем
   #Temp := #Temp AND #Temp_In;                  // Изменившиеся биты обнуляеми а не изменившиеся с последнего скана биты запоминаем 
   #Slot.Value := #Slot.Value OR #Temp;                 // Формируем выход 
   #Slot.Value_Last_Scan := #Temp_In;                   // Запоминаем текущее значение как значение последнего скана

   // При включенной симуляции заменяем исходное значение на Sim_Value
   #Slot.Value := (#Slot.Sim_En AND #Slot.Sim_Value) OR ((NOT #Slot.Sim_En) AND #Slot.Value);

   FOR #i := 0 TO 7 DO
     #Slot.Pins[#i] := "GetBitByte"(Data := #Slot.Value,
                                    pos := #i);
   END_FOR;
END_FUNCTION_BLOCK

FUNCTION_BLOCK "Put_DO32"   // FB5, SCL
TITLE = 'Puts 32-bit DO module data to Q-output'
{ S7_Optimized_Access := 'FALSE' }
NAME : PutDO32
VERSION : 1.0
   VAR_OUTPUT
      Out : DWord;
   END_VAR
   VAR
      Slot : Struct
         Data_to_out : DWord;   // block input data
         Pins : Array[0..31] of Bool;   // hardware pins (accordance byte order)
         UsePinsAsInput : Bool := TRUE;   // true if Pins owerride Data_to_output
         Invert_En : DWord;   // invert mask
         Output_En : DWord;   // enable output mask
         Sim_En : DWord;   // simulate enable mask
         Sim_Value : DWord;   // simulate value
         Value : DWord;   // Result after enable and filtering
      END_STRUCT;
   END_VAR
   VAR_TEMP
      Temp : DWord;
      i : Int;
      Hi : Word;
      Lo : Word;
   END_VAR
BEGIN


   IF #Slot.UsePinsAsInput THEN
     FOR #i := 0 TO 7 DO
       "SetBitWord"(pos := #i,
                    value := #Slot.Pins[#i + 24],
                    Data := #Lo);
       "SetBitWord"(pos := #i + 8,
                    value := #Slot.Pins[#i + 16],
                    Data := #Lo);
       "SetBitWord"(pos := #i,
                    value := #Slot.Pins[#i + 8],
                    Data := #Hi);
       "SetBitWord"(pos := #i + 8,
                    value := #Slot.Pins[#i],
                    Data := #Hi);
     END_FOR;
     #Slot.Data_to_out := #Hi * 16#10000 + #Lo;
   END_IF;

   #Temp := #Slot.Data_to_out XOR #Slot.Invert_En; // Инвертирование сигналов  
   #Slot.Value := #Temp AND #Slot.Output_En;           // Проходят  только разрешенные синалы 

   // При включенной симуляции заменяем исходное значение на Sim_Value
   #Out := (#Slot.Sim_En AND #Slot.Sim_Value) OR ((NOT #Slot.Sim_En) AND #Slot.Value);
END_FUNCTION_BLOCK

FUNCTION_BLOCK "Put_DO16"   // FB6, SCL
TITLE = 'Puts 16-bit DO module data to Q-output'
{ S7_Optimized_Access := 'TRUE' }
NAME : PutDO16
VERSION : 1.0
   VAR_OUTPUT
      Out : Word;
   END_VAR
   VAR
      Slot : Struct
         Data_to_out : Word;   // block input data
         Pins : Array[0..15] of Bool;   // hardware pins (accordance byte order)
         UsePinsAsInput : Bool := TRUE;   // true if Pins owerride Data_to_output
         Invert_En : Word;   // invert mask
         Output_En_out : Word;   // enable output mask
         Sim_En_out : Word;   // simulate enable mask
         Sim_Value_out : Word;   // simulate value
         Value : Word;   // Result after enable and filtering
      END_STRUCT;
   END_VAR
   VAR_TEMP
      Temp : Word;
      i : Int;
   END_VAR
BEGIN

   (*#Slot.Output_En_out:= 16#1111;*)
   #Slot.UsePinsAsInput := true;
   IF #Slot.UsePinsAsInput THEN
     FOR #i := 0 TO 7 DO
       "SetBitWord"(pos := #i,
                    value := #Slot.Pins[#i + 8],
                    Data := #Slot.Data_to_out);
       "SetBitWord"(pos := #i + 8,
                    value := #Slot.Pins[#i],
                    Data := #Slot.Data_to_out);
     END_FOR;
   END_IF;

   #Temp := #Slot.Data_to_out XOR #Slot.Invert_En; // Инвертирование сигналов  
   #Slot.Value := #Temp AND #Slot.Output_En_out;           // Проходят  только разрешенные синалы 

   // При включенной симуляции заменяем исходное значение на Sim_Value
   #Out := (#Slot.Sim_En_out AND #Slot.Sim_Value_out) OR ((NOT #Slot.Sim_En_out) AND #Slot.Value);
END_FUNCTION_BLOCK

// folder: Modbus

FUNCTION "Write_to_MB" : Void   // FC8, SCL
{ S7_Optimized_Access := 'TRUE' }
VERSION : 0.1
BEGIN
   //***************Перекладывание для ВУ **************
   "Modbus_Buffer".Lamp_1_on_door := "Fire";
   "Modbus_Buffer".Spark_1_to_on :="Spark_on";
   "Modbus_Buffer".Man_on := "Torche_DB".Man_fakel;
   "Modbus_Buffer".DO_Alarm := "Torche_DB".DO_Alarm;
   "Modbus_Buffer".Valve_to_open_lamp_on := "Torche_DB".Valve_to_open;


   "Modbus_Buffer".Time_Venting := "Torche_DB".Signal_Torche.Time_vent_g;
   "Modbus_Buffer".Time_firing := "Torche_DB".Signal_Torche.Time_firing_g;
   "Modbus_Buffer".Time_spark_on := "Torche_DB".Signal_Torche.Time_spark_on_g;
   "Modbus_Buffer".Time_spark_off:= "Torche_DB".Signal_Torche.Time_spark_off_g;
   "Modbus_Buffer".Time_stabil := "Torche_DB".Signal_Torche.Time_stabiliz_g;
   "Modbus_Buffer".Time_after_alarm := "Torche_DB".Signal_Torche.Time_after_alm_g;
   "Modbus_Buffer".Time_after_stop := "Torche_DB".Signal_Torche.Time_stop_fire_g;

   "Modbus_Buffer".Temp_Fire := "Temp_gorelka".Signal_AI.HH_Lim ;
   "Modbus_Buffer".Scal_max := "Temp_gorelka".Signal_AI.Scal_Max_Eu;
   "Modbus_Buffer".Scal_min := "Temp_gorelka".Signal_AI.Scal_Min_Eu;
   "Modbus_Buffer".Temp_ACP := "Temp_gorelka".Signal_AI.Acp;

   "Modbus_Buffer".Temp_Fire_2 := "temp_gorelka_2".Signal_AI.HH_Lim;
   "Modbus_Buffer".Scal_max_2 := "temp_gorelka_2".Signal_AI.Scal_Max_Eu;
   "Modbus_Buffer".Scal_min_2 := "temp_gorelka_2".Signal_AI.Scal_Min_Eu;
   "Modbus_Buffer".Temp_ACP_2 := "temp_gorelka_2".Signal_AI.Acp;
END_FUNCTION

FUNCTION "Read_from_MB" : Void   // FC10, SCL
{ S7_Optimized_Access := 'TRUE' }
VERSION : 0.1
BEGIN
   //**********Запись времени сверху по Modbus******************

